DATA_BLOCK "InstEmDataHmi"   // DB44
TITLE = Instanz von FB EnergyMeterDataToHmi / Instance of FB instance of FB EnergyMeterDataToHmi
AUTHOR : SICAR
FAMILY : Energy
VERSION : 1.0
// Energy meter HMI
// stored: InstanceOfName LSicar_EnMeterDataToHmi, InstanceOfType FB
"LSicar_EnMeterDataToHmi"
   // VAR_INPUT
   //    energyMeter01Visu { ExternalAccessible := 'False'; ExternalVisible := 'False'; ExternalWritable := 'False'} : "LSicar_typeEnMeterVisuStruct";
   //    energyMeter02Visu { ExternalAccessible := 'False'; ExternalVisible := 'False'; ExternalWritable := 'False'} : "LSicar_typeEnMeterVisuStruct";
   //    energyMeter03Visu { ExternalAccessible := 'False'; ExternalVisible := 'False'; ExternalWritable := 'False'} : "LSicar_typeEnMeterVisuStruct";
   //    energyMeter04Visu { ExternalAccessible := 'False'; ExternalVisible := 'False'; ExternalWritable := 'False'} : "LSicar_typeEnMeterVisuStruct";
   //    energyMeter05Visu { ExternalAccessible := 'False'; ExternalVisible := 'False'; ExternalWritable := 'False'} : "LSicar_typeEnMeterVisuStruct";
   //    energyMeter06Visu { ExternalAccessible := 'False'; ExternalVisible := 'False'; ExternalWritable := 'False'} : "LSicar_typeEnMeterVisuStruct";
   //    energyMeter07Visu { ExternalAccessible := 'False'; ExternalVisible := 'False'; ExternalWritable := 'False'} : "LSicar_typeEnMeterVisuStruct";
   //    energyMeter08Visu { ExternalAccessible := 'False'; ExternalVisible := 'False'; ExternalWritable := 'False'} : "LSicar_typeEnMeterVisuStruct";
   // END_VAR
   // VAR
   //    statEmIndex : Int := 1;
   //    statEmData : "LSicar_typeEnMeterVisuStruct";
   //    statResetMinMaxAll : Bool := FALSE;
   //    statResetMinMax : Array[0..8] of Bool;
   //    statResetEnCounterAll : Bool := FALSE;
   //    statResetEnCounter : Array[0..8] of Bool;
   // END_VAR
BEGIN
   energyMeter01Visu.uL1L2 := 480.6464;
   energyMeter01Visu.uL2L3 := 479.3329;
   energyMeter01Visu.uL3L1 := 482.4024;
   energyMeter01Visu.uL1 := 277.0244;
   energyMeter01Visu.uL2 := 283.0648;
   energyMeter01Visu.uL3 := 272.9026;
   energyMeter01Visu.uL1L2Min := 470.1363;
   energyMeter01Visu.uL2L3Min := 469.0945;
   energyMeter01Visu.uL3L1Min := 472.4617;
   energyMeter01Visu.uL1Min := 271.5103;
   energyMeter01Visu.uL2Min := 277.1332;
   energyMeter01Visu.uL3Min := 267.6445;
   energyMeter01Visu.uL1L2Max := 486.0269;
   energyMeter01Visu.uL2L3Max := 484.8441;
   energyMeter01Visu.uL3L1Max := 487.8807;
   energyMeter01Visu.uL1Max := 280.1993;
   energyMeter01Visu.uL2Max := 286.2231;
   energyMeter01Visu.uL3Max := 276.0547;
   energyMeter01Visu.uPhPhAverage := 480.7939;
   energyMeter01Visu.uPhNaverage := 277.6639;
   energyMeter01Visu.uPhPhAverageMin := 470.5642;
   energyMeter01Visu.uPhNaverageMin := 272.105;
   energyMeter01Visu.uPhPhAverageMax := 486.2456;
   energyMeter01Visu.uPhNaverageMax := 280.8176;
   energyMeter01Visu.iL1 := 0.6297245;
   energyMeter01Visu.iL2 := 0.4116209;
   energyMeter01Visu.iL3 := 0.4021624;
   energyMeter01Visu.iL1Min := 0.5503862;
   energyMeter01Visu.iL2Min := 0.3512777;
   energyMeter01Visu.iL3Min := 0.3410119;
   energyMeter01Visu.iL1Max := 2.701323;
   energyMeter01Visu.iL2Max := 2.376321;
   energyMeter01Visu.iL3Max := 1.768756;
   energyMeter01Visu.iAverage := 0.4811693;
   energyMeter01Visu.iAverageMin := 0.4219982;
   energyMeter01Visu.iAverageMax := 2.194234;
   energyMeter01Visu.f := 59.99327;
   energyMeter01Visu.fMin := 59.9567;
   energyMeter01Visu.fMax := 60.07609;
   energyMeter01Visu.sTotal := 400.7156;
   energyMeter01Visu.sTotalMin := 349.7767;
   energyMeter01Visu.sTotalMax := 1823.43;
   energyMeter01Visu.pTotal := 277.3849;
   energyMeter01Visu.pTotalMin := 220.7085;
   energyMeter01Visu.pTotalMax := 670.0833;
   energyMeter01Visu.qTotal := -19.24654;
   energyMeter01Visu.qTotalMin := -422.0206;
   energyMeter01Visu.qTotalMax := -5.418034;
   energyMeter01Visu.cosL1 := 0.8610036;
   energyMeter01Visu.cosL1Min := 0.3576268;
   energyMeter01Visu.cosL1Max := 0.9157406;
   energyMeter01Visu.cosL2 := 0.5061908;
   energyMeter01Visu.cosL2Min := 0.05827232;
   energyMeter01Visu.cosL2Max := 0.7094496;
   energyMeter01Visu.cosL3 := 0.6214478;
   energyMeter01Visu.cosL3Min := 0.1665398;
   energyMeter01Visu.cosL3Max := 0.7301649;
   energyMeter01Visu.cosAverage := 0.6922238;
   energyMeter01Visu.cosAverageMin := 0.2474333;
   energyMeter01Visu.cosAverageMax := 0.7716895;
   energyMeter01Visu.sL1 := 174.449;
   energyMeter01Visu.sL2 := 116.5154;
   energyMeter01Visu.sL3 := 109.7511;
   energyMeter01Visu.sL1Min := 151.7066;
   energyMeter01Visu.sL2Min := 99.03358;
   energyMeter01Visu.sL3Min := 92.7289;
   energyMeter01Visu.sL1Max := 744.3881;
   energyMeter01Visu.sL2Max := 669.9091;
   energyMeter01Visu.sL3Max := 480.3434;
   energyMeter01Visu.pL1 := 150.2012;
   energyMeter01Visu.pL2 := 58.97903;
   energyMeter01Visu.pL3 := 68.20461;
   energyMeter01Visu.pL1Min := 127.6866;
   energyMeter01Visu.pL2Min := 20.87;
   energyMeter01Visu.pL3Min := 52.5906;
   energyMeter01Visu.pL1Max := 281.8818;
   energyMeter01Visu.pL2Max := 194.1828;
   energyMeter01Visu.pL3Max := 220.8245;
   energyMeter01Visu.qL1 := -4.041785;
   energyMeter01Visu.qL2 := 41.25737;
   energyMeter01Visu.qL3 := -56.46213;
   energyMeter01Visu.qL1Min := -144.4171;
   energyMeter01Visu.qL2Min := -98.00859;
   energyMeter01Visu.qL3Min := -198.8008;
   energyMeter01Visu.qL1Max := 28.71266;
   energyMeter01Visu.qL2Max := 50.3845;
   energyMeter01Visu.qL3Max := -53.43742;
   energyMeter01Visu.eActiveRate1Import := 736796.1;
   energyMeter01Visu.eActiveRate2Import := 0.0;
   energyMeter01Visu.eActiveRate1Export := 0.0002530577;
   energyMeter01Visu.eActiveRate2Export := 0.0;
   energyMeter01Visu.eReactiveRate1Import := 5676.457;
   energyMeter01Visu.eReactiveRate2Import := 0.0;
   energyMeter01Visu.eReactiveRate1Export := 293593.3;
   energyMeter01Visu.eReactiveRate2Export := 0.0;
   energyMeter01Visu.eApparentRate1Import := 1470773.0;
   energyMeter01Visu.eApparentRate2Import := 0.0;
   energyMeter01Visu.rTimeDataEnergy := DTL#1970-01-01-00:00:00;
   energyMeter01Visu.rTimeDataValue := DTL#1970-01-01-00:00:00;
   energyMeter01Visu.uPhPhMod := 16#0000;
   energyMeter01Visu.uPhNmod := 16#0000;
   energyMeter01Visu.iMod := 16#0000;
   energyMeter01Visu.sMod := 16#0000;
   energyMeter01Visu.pMod := 16#0000;
   energyMeter01Visu.qMod := 16#0000;
   energyMeter01Visu.eMod := 16#0000;
   energyMeter01Visu.fMod := 16#0000;
   energyMeter01Visu.cosMod := 16#0000;
   energyMeter01Visu.calculateValue1 := 16#0000;
   energyMeter01Visu.calculateValue2 := 16#0000;
   energyMeter01Visu.calculateValue3 := 16#0000;
   energyMeter01Visu.calculateValue4 := 16#0000;
   energyMeter01Visu.calculateValue5 := 16#0000;
   energyMeter01Visu.calculateValue6 := 16#0000;
   energyMeter01Visu.energyMeterUnit := 16#0000;
   energyMeter01Visu.restStartAuto := FALSE;
   energyMeter01Visu.readValue := FALSE;
   energyMeter01Visu.connectionType := 0;
   energyMeter01Visu.driverError := 0;
   energyMeter02Visu.uL1L2 := 0.0;
   energyMeter02Visu.uL2L3 := 0.0;
   energyMeter02Visu.uL3L1 := 0.0;
   energyMeter02Visu.uL1 := 0.0;
   energyMeter02Visu.uL2 := 0.0;
   energyMeter02Visu.uL3 := 0.0;
   energyMeter02Visu.uL1L2Min := 0.0;
   energyMeter02Visu.uL2L3Min := 0.0;
   energyMeter02Visu.uL3L1Min := 0.0;
   energyMeter02Visu.uL1Min := 0.0;
   energyMeter02Visu.uL2Min := 0.0;
   energyMeter02Visu.uL3Min := 0.0;
   energyMeter02Visu.uL1L2Max := 0.0;
   energyMeter02Visu.uL2L3Max := 0.0;
   energyMeter02Visu.uL3L1Max := 0.0;
   energyMeter02Visu.uL1Max := 0.0;
   energyMeter02Visu.uL2Max := 0.0;
   energyMeter02Visu.uL3Max := 0.0;
   energyMeter02Visu.uPhPhAverage := 0.0;
   energyMeter02Visu.uPhNaverage := 0.0;
   energyMeter02Visu.uPhPhAverageMin := 0.0;
   energyMeter02Visu.uPhNaverageMin := 0.0;
   energyMeter02Visu.uPhPhAverageMax := 0.0;
   energyMeter02Visu.uPhNaverageMax := 0.0;
   energyMeter02Visu.iL1 := 0.0;
   energyMeter02Visu.iL2 := 0.0;
   energyMeter02Visu.iL3 := 0.0;
   energyMeter02Visu.iL1Min := 0.0;
   energyMeter02Visu.iL2Min := 0.0;
   energyMeter02Visu.iL3Min := 0.0;
   energyMeter02Visu.iL1Max := 0.0;
   energyMeter02Visu.iL2Max := 0.0;
   energyMeter02Visu.iL3Max := 0.0;
   energyMeter02Visu.iAverage := 0.0;
   energyMeter02Visu.iAverageMin := 0.0;
   energyMeter02Visu.iAverageMax := 0.0;
   energyMeter02Visu.f := 0.0;
   energyMeter02Visu.fMin := 0.0;
   energyMeter02Visu.fMax := 0.0;
   energyMeter02Visu.sTotal := 0.0;
   energyMeter02Visu.sTotalMin := 0.0;
   energyMeter02Visu.sTotalMax := 0.0;
   energyMeter02Visu.pTotal := 0.0;
   energyMeter02Visu.pTotalMin := 0.0;
   energyMeter02Visu.pTotalMax := 0.0;
   energyMeter02Visu.qTotal := 0.0;
   energyMeter02Visu.qTotalMin := 0.0;
   energyMeter02Visu.qTotalMax := 0.0;
   energyMeter02Visu.cosL1 := 0.0;
   energyMeter02Visu.cosL1Min := 0.0;
   energyMeter02Visu.cosL1Max := 0.0;
   energyMeter02Visu.cosL2 := 0.0;
   energyMeter02Visu.cosL2Min := 0.0;
   energyMeter02Visu.cosL2Max := 0.0;
   energyMeter02Visu.cosL3 := 0.0;
   energyMeter02Visu.cosL3Min := 0.0;
   energyMeter02Visu.cosL3Max := 0.0;
   energyMeter02Visu.cosAverage := 0.0;
   energyMeter02Visu.cosAverageMin := 0.0;
   energyMeter02Visu.cosAverageMax := 0.0;
   energyMeter02Visu.sL1 := 0.0;
   energyMeter02Visu.sL2 := 0.0;
   energyMeter02Visu.sL3 := 0.0;
   energyMeter02Visu.sL1Min := 0.0;
   energyMeter02Visu.sL2Min := 0.0;
   energyMeter02Visu.sL3Min := 0.0;
   energyMeter02Visu.sL1Max := 0.0;
   energyMeter02Visu.sL2Max := 0.0;
   energyMeter02Visu.sL3Max := 0.0;
   energyMeter02Visu.pL1 := 0.0;
   energyMeter02Visu.pL2 := 0.0;
   energyMeter02Visu.pL3 := 0.0;
   energyMeter02Visu.pL1Min := 0.0;
   energyMeter02Visu.pL2Min := 0.0;
   energyMeter02Visu.pL3Min := 0.0;
   energyMeter02Visu.pL1Max := 0.0;
   energyMeter02Visu.pL2Max := 0.0;
   energyMeter02Visu.pL3Max := 0.0;
   energyMeter02Visu.qL1 := 0.0;
   energyMeter02Visu.qL2 := 0.0;
   energyMeter02Visu.qL3 := 0.0;
   energyMeter02Visu.qL1Min := 0.0;
   energyMeter02Visu.qL2Min := 0.0;
   energyMeter02Visu.qL3Min := 0.0;
   energyMeter02Visu.qL1Max := 0.0;
   energyMeter02Visu.qL2Max := 0.0;
   energyMeter02Visu.qL3Max := 0.0;
   energyMeter02Visu.eActiveRate1Import := 0.0;
   energyMeter02Visu.eActiveRate2Import := 0.0;
   energyMeter02Visu.eActiveRate1Export := 0.0;
   energyMeter02Visu.eActiveRate2Export := 0.0;
   energyMeter02Visu.eReactiveRate1Import := 0.0;
   energyMeter02Visu.eReactiveRate2Import := 0.0;
   energyMeter02Visu.eReactiveRate1Export := 0.0;
   energyMeter02Visu.eReactiveRate2Export := 0.0;
   energyMeter02Visu.eApparentRate1Import := 0.0;
   energyMeter02Visu.eApparentRate2Import := 0.0;
   energyMeter02Visu.rTimeDataEnergy := DTL#1970-01-01-00:00:00;
   energyMeter02Visu.rTimeDataValue := DTL#1970-01-01-00:00:00;
   energyMeter02Visu.uPhPhMod := 16#0000;
   energyMeter02Visu.uPhNmod := 16#0000;
   energyMeter02Visu.iMod := 16#0000;
   energyMeter02Visu.sMod := 16#0000;
   energyMeter02Visu.pMod := 16#0000;
   energyMeter02Visu.qMod := 16#0000;
   energyMeter02Visu.eMod := 16#0000;
   energyMeter02Visu.fMod := 16#0000;
   energyMeter02Visu.cosMod := 16#0000;
   energyMeter02Visu.calculateValue1 := 16#0000;
   energyMeter02Visu.calculateValue2 := 16#0000;
   energyMeter02Visu.calculateValue3 := 16#0000;
   energyMeter02Visu.calculateValue4 := 16#0000;
   energyMeter02Visu.calculateValue5 := 16#0000;
   energyMeter02Visu.calculateValue6 := 16#0000;
   energyMeter02Visu.energyMeterUnit := 16#0000;
   energyMeter02Visu.restStartAuto := FALSE;
   energyMeter02Visu.readValue := FALSE;
   energyMeter02Visu.connectionType := 0;
   energyMeter02Visu.driverError := 0;
   energyMeter03Visu.uL1L2 := 0.0;
   energyMeter03Visu.uL2L3 := 0.0;
   energyMeter03Visu.uL3L1 := 0.0;
   energyMeter03Visu.uL1 := 0.0;
   energyMeter03Visu.uL2 := 0.0;
   energyMeter03Visu.uL3 := 0.0;
   energyMeter03Visu.uL1L2Min := 0.0;
   energyMeter03Visu.uL2L3Min := 0.0;
   energyMeter03Visu.uL3L1Min := 0.0;
   energyMeter03Visu.uL1Min := 0.0;
   energyMeter03Visu.uL2Min := 0.0;
   energyMeter03Visu.uL3Min := 0.0;
   energyMeter03Visu.uL1L2Max := 0.0;
   energyMeter03Visu.uL2L3Max := 0.0;
   energyMeter03Visu.uL3L1Max := 0.0;
   energyMeter03Visu.uL1Max := 0.0;
   energyMeter03Visu.uL2Max := 0.0;
   energyMeter03Visu.uL3Max := 0.0;
   energyMeter03Visu.uPhPhAverage := 0.0;
   energyMeter03Visu.uPhNaverage := 0.0;
   energyMeter03Visu.uPhPhAverageMin := 0.0;
   energyMeter03Visu.uPhNaverageMin := 0.0;
   energyMeter03Visu.uPhPhAverageMax := 0.0;
   energyMeter03Visu.uPhNaverageMax := 0.0;
   energyMeter03Visu.iL1 := 0.0;
   energyMeter03Visu.iL2 := 0.0;
   energyMeter03Visu.iL3 := 0.0;
   energyMeter03Visu.iL1Min := 0.0;
   energyMeter03Visu.iL2Min := 0.0;
   energyMeter03Visu.iL3Min := 0.0;
   energyMeter03Visu.iL1Max := 0.0;
   energyMeter03Visu.iL2Max := 0.0;
   energyMeter03Visu.iL3Max := 0.0;
   energyMeter03Visu.iAverage := 0.0;
   energyMeter03Visu.iAverageMin := 0.0;
   energyMeter03Visu.iAverageMax := 0.0;
   energyMeter03Visu.f := 0.0;
   energyMeter03Visu.fMin := 0.0;
   energyMeter03Visu.fMax := 0.0;
   energyMeter03Visu.sTotal := 0.0;
   energyMeter03Visu.sTotalMin := 0.0;
   energyMeter03Visu.sTotalMax := 0.0;
   energyMeter03Visu.pTotal := 0.0;
   energyMeter03Visu.pTotalMin := 0.0;
   energyMeter03Visu.pTotalMax := 0.0;
   energyMeter03Visu.qTotal := 0.0;
   energyMeter03Visu.qTotalMin := 0.0;
   energyMeter03Visu.qTotalMax := 0.0;
   energyMeter03Visu.cosL1 := 0.0;
   energyMeter03Visu.cosL1Min := 0.0;
   energyMeter03Visu.cosL1Max := 0.0;
   energyMeter03Visu.cosL2 := 0.0;
   energyMeter03Visu.cosL2Min := 0.0;
   energyMeter03Visu.cosL2Max := 0.0;
   energyMeter03Visu.cosL3 := 0.0;
   energyMeter03Visu.cosL3Min := 0.0;
   energyMeter03Visu.cosL3Max := 0.0;
   energyMeter03Visu.cosAverage := 0.0;
   energyMeter03Visu.cosAverageMin := 0.0;
   energyMeter03Visu.cosAverageMax := 0.0;
   energyMeter03Visu.sL1 := 0.0;
   energyMeter03Visu.sL2 := 0.0;
   energyMeter03Visu.sL3 := 0.0;
   energyMeter03Visu.sL1Min := 0.0;
   energyMeter03Visu.sL2Min := 0.0;
   energyMeter03Visu.sL3Min := 0.0;
   energyMeter03Visu.sL1Max := 0.0;
   energyMeter03Visu.sL2Max := 0.0;
   energyMeter03Visu.sL3Max := 0.0;
   energyMeter03Visu.pL1 := 0.0;
   energyMeter03Visu.pL2 := 0.0;
   energyMeter03Visu.pL3 := 0.0;
   energyMeter03Visu.pL1Min := 0.0;
   energyMeter03Visu.pL2Min := 0.0;
   energyMeter03Visu.pL3Min := 0.0;
   energyMeter03Visu.pL1Max := 0.0;
   energyMeter03Visu.pL2Max := 0.0;
   energyMeter03Visu.pL3Max := 0.0;
   energyMeter03Visu.qL1 := 0.0;
   energyMeter03Visu.qL2 := 0.0;
   energyMeter03Visu.qL3 := 0.0;
   energyMeter03Visu.qL1Min := 0.0;
   energyMeter03Visu.qL2Min := 0.0;
   energyMeter03Visu.qL3Min := 0.0;
   energyMeter03Visu.qL1Max := 0.0;
   energyMeter03Visu.qL2Max := 0.0;
   energyMeter03Visu.qL3Max := 0.0;
   energyMeter03Visu.eActiveRate1Import := 0.0;
   energyMeter03Visu.eActiveRate2Import := 0.0;
   energyMeter03Visu.eActiveRate1Export := 0.0;
   energyMeter03Visu.eActiveRate2Export := 0.0;
   energyMeter03Visu.eReactiveRate1Import := 0.0;
   energyMeter03Visu.eReactiveRate2Import := 0.0;
   energyMeter03Visu.eReactiveRate1Export := 0.0;
   energyMeter03Visu.eReactiveRate2Export := 0.0;
   energyMeter03Visu.eApparentRate1Import := 0.0;
   energyMeter03Visu.eApparentRate2Import := 0.0;
   energyMeter03Visu.rTimeDataEnergy := DTL#1970-01-01-00:00:00;
   energyMeter03Visu.rTimeDataValue := DTL#1970-01-01-00:00:00;
   energyMeter03Visu.uPhPhMod := 16#0000;
   energyMeter03Visu.uPhNmod := 16#0000;
   energyMeter03Visu.iMod := 16#0000;
   energyMeter03Visu.sMod := 16#0000;
   energyMeter03Visu.pMod := 16#0000;
   energyMeter03Visu.qMod := 16#0000;
   energyMeter03Visu.eMod := 16#0000;
   energyMeter03Visu.fMod := 16#0000;
   energyMeter03Visu.cosMod := 16#0000;
   energyMeter03Visu.calculateValue1 := 16#0000;
   energyMeter03Visu.calculateValue2 := 16#0000;
   energyMeter03Visu.calculateValue3 := 16#0000;
   energyMeter03Visu.calculateValue4 := 16#0000;
   energyMeter03Visu.calculateValue5 := 16#0000;
   energyMeter03Visu.calculateValue6 := 16#0000;
   energyMeter03Visu.energyMeterUnit := 16#0000;
   energyMeter03Visu.restStartAuto := FALSE;
   energyMeter03Visu.readValue := FALSE;
   energyMeter03Visu.connectionType := 0;
   energyMeter03Visu.driverError := 0;
   energyMeter04Visu.uL1L2 := 0.0;
   energyMeter04Visu.uL2L3 := 0.0;
   energyMeter04Visu.uL3L1 := 0.0;
   energyMeter04Visu.uL1 := 0.0;
   energyMeter04Visu.uL2 := 0.0;
   energyMeter04Visu.uL3 := 0.0;
   energyMeter04Visu.uL1L2Min := 0.0;
   energyMeter04Visu.uL2L3Min := 0.0;
   energyMeter04Visu.uL3L1Min := 0.0;
   energyMeter04Visu.uL1Min := 0.0;
   energyMeter04Visu.uL2Min := 0.0;
   energyMeter04Visu.uL3Min := 0.0;
   energyMeter04Visu.uL1L2Max := 0.0;
   energyMeter04Visu.uL2L3Max := 0.0;
   energyMeter04Visu.uL3L1Max := 0.0;
   energyMeter04Visu.uL1Max := 0.0;
   energyMeter04Visu.uL2Max := 0.0;
   energyMeter04Visu.uL3Max := 0.0;
   energyMeter04Visu.uPhPhAverage := 0.0;
   energyMeter04Visu.uPhNaverage := 0.0;
   energyMeter04Visu.uPhPhAverageMin := 0.0;
   energyMeter04Visu.uPhNaverageMin := 0.0;
   energyMeter04Visu.uPhPhAverageMax := 0.0;
   energyMeter04Visu.uPhNaverageMax := 0.0;
   energyMeter04Visu.iL1 := 0.0;
   energyMeter04Visu.iL2 := 0.0;
   energyMeter04Visu.iL3 := 0.0;
   energyMeter04Visu.iL1Min := 0.0;
   energyMeter04Visu.iL2Min := 0.0;
   energyMeter04Visu.iL3Min := 0.0;
   energyMeter04Visu.iL1Max := 0.0;
   energyMeter04Visu.iL2Max := 0.0;
   energyMeter04Visu.iL3Max := 0.0;
   energyMeter04Visu.iAverage := 0.0;
   energyMeter04Visu.iAverageMin := 0.0;
   energyMeter04Visu.iAverageMax := 0.0;
   energyMeter04Visu.f := 0.0;
   energyMeter04Visu.fMin := 0.0;
   energyMeter04Visu.fMax := 0.0;
   energyMeter04Visu.sTotal := 0.0;
   energyMeter04Visu.sTotalMin := 0.0;
   energyMeter04Visu.sTotalMax := 0.0;
   energyMeter04Visu.pTotal := 0.0;
   energyMeter04Visu.pTotalMin := 0.0;
   energyMeter04Visu.pTotalMax := 0.0;
   energyMeter04Visu.qTotal := 0.0;
   energyMeter04Visu.qTotalMin := 0.0;
   energyMeter04Visu.qTotalMax := 0.0;
   energyMeter04Visu.cosL1 := 0.0;
   energyMeter04Visu.cosL1Min := 0.0;
   energyMeter04Visu.cosL1Max := 0.0;
   energyMeter04Visu.cosL2 := 0.0;
   energyMeter04Visu.cosL2Min := 0.0;
   energyMeter04Visu.cosL2Max := 0.0;
   energyMeter04Visu.cosL3 := 0.0;
   energyMeter04Visu.cosL3Min := 0.0;
   energyMeter04Visu.cosL3Max := 0.0;
   energyMeter04Visu.cosAverage := 0.0;
   energyMeter04Visu.cosAverageMin := 0.0;
   energyMeter04Visu.cosAverageMax := 0.0;
   energyMeter04Visu.sL1 := 0.0;
   energyMeter04Visu.sL2 := 0.0;
   energyMeter04Visu.sL3 := 0.0;
   energyMeter04Visu.sL1Min := 0.0;
   energyMeter04Visu.sL2Min := 0.0;
   energyMeter04Visu.sL3Min := 0.0;
   energyMeter04Visu.sL1Max := 0.0;
   energyMeter04Visu.sL2Max := 0.0;
   energyMeter04Visu.sL3Max := 0.0;
   energyMeter04Visu.pL1 := 0.0;
   energyMeter04Visu.pL2 := 0.0;
   energyMeter04Visu.pL3 := 0.0;
   energyMeter04Visu.pL1Min := 0.0;
   energyMeter04Visu.pL2Min := 0.0;
   energyMeter04Visu.pL3Min := 0.0;
   energyMeter04Visu.pL1Max := 0.0;
   energyMeter04Visu.pL2Max := 0.0;
   energyMeter04Visu.pL3Max := 0.0;
   energyMeter04Visu.qL1 := 0.0;
   energyMeter04Visu.qL2 := 0.0;
   energyMeter04Visu.qL3 := 0.0;
   energyMeter04Visu.qL1Min := 0.0;
   energyMeter04Visu.qL2Min := 0.0;
   energyMeter04Visu.qL3Min := 0.0;
   energyMeter04Visu.qL1Max := 0.0;
   energyMeter04Visu.qL2Max := 0.0;
   energyMeter04Visu.qL3Max := 0.0;
   energyMeter04Visu.eActiveRate1Import := 0.0;
   energyMeter04Visu.eActiveRate2Import := 0.0;
   energyMeter04Visu.eActiveRate1Export := 0.0;
   energyMeter04Visu.eActiveRate2Export := 0.0;
   energyMeter04Visu.eReactiveRate1Import := 0.0;
   energyMeter04Visu.eReactiveRate2Import := 0.0;
   energyMeter04Visu.eReactiveRate1Export := 0.0;
   energyMeter04Visu.eReactiveRate2Export := 0.0;
   energyMeter04Visu.eApparentRate1Import := 0.0;
   energyMeter04Visu.eApparentRate2Import := 0.0;
   energyMeter04Visu.rTimeDataEnergy := DTL#1970-01-01-00:00:00;
   energyMeter04Visu.rTimeDataValue := DTL#1970-01-01-00:00:00;
   energyMeter04Visu.uPhPhMod := 16#0000;
   energyMeter04Visu.uPhNmod := 16#0000;
   energyMeter04Visu.iMod := 16#0000;
   energyMeter04Visu.sMod := 16#0000;
   energyMeter04Visu.pMod := 16#0000;
   energyMeter04Visu.qMod := 16#0000;
   energyMeter04Visu.eMod := 16#0000;
   energyMeter04Visu.fMod := 16#0000;
   energyMeter04Visu.cosMod := 16#0000;
   energyMeter04Visu.calculateValue1 := 16#0000;
   energyMeter04Visu.calculateValue2 := 16#0000;
   energyMeter04Visu.calculateValue3 := 16#0000;
   energyMeter04Visu.calculateValue4 := 16#0000;
   energyMeter04Visu.calculateValue5 := 16#0000;
   energyMeter04Visu.calculateValue6 := 16#0000;
   energyMeter04Visu.energyMeterUnit := 16#0000;
   energyMeter04Visu.restStartAuto := FALSE;
   energyMeter04Visu.readValue := FALSE;
   energyMeter04Visu.connectionType := 0;
   energyMeter04Visu.driverError := 0;
   energyMeter05Visu.uL1L2 := 0.0;
   energyMeter05Visu.uL2L3 := 0.0;
   energyMeter05Visu.uL3L1 := 0.0;
   energyMeter05Visu.uL1 := 0.0;
   energyMeter05Visu.uL2 := 0.0;
   energyMeter05Visu.uL3 := 0.0;
   energyMeter05Visu.uL1L2Min := 0.0;
   energyMeter05Visu.uL2L3Min := 0.0;
   energyMeter05Visu.uL3L1Min := 0.0;
   energyMeter05Visu.uL1Min := 0.0;
   energyMeter05Visu.uL2Min := 0.0;
   energyMeter05Visu.uL3Min := 0.0;
   energyMeter05Visu.uL1L2Max := 0.0;
   energyMeter05Visu.uL2L3Max := 0.0;
   energyMeter05Visu.uL3L1Max := 0.0;
   energyMeter05Visu.uL1Max := 0.0;
   energyMeter05Visu.uL2Max := 0.0;
   energyMeter05Visu.uL3Max := 0.0;
   energyMeter05Visu.uPhPhAverage := 0.0;
   energyMeter05Visu.uPhNaverage := 0.0;
   energyMeter05Visu.uPhPhAverageMin := 0.0;
   energyMeter05Visu.uPhNaverageMin := 0.0;
   energyMeter05Visu.uPhPhAverageMax := 0.0;
   energyMeter05Visu.uPhNaverageMax := 0.0;
   energyMeter05Visu.iL1 := 0.0;
   energyMeter05Visu.iL2 := 0.0;
   energyMeter05Visu.iL3 := 0.0;
   energyMeter05Visu.iL1Min := 0.0;
   energyMeter05Visu.iL2Min := 0.0;
   energyMeter05Visu.iL3Min := 0.0;
   energyMeter05Visu.iL1Max := 0.0;
   energyMeter05Visu.iL2Max := 0.0;
   energyMeter05Visu.iL3Max := 0.0;
   energyMeter05Visu.iAverage := 0.0;
   energyMeter05Visu.iAverageMin := 0.0;
   energyMeter05Visu.iAverageMax := 0.0;
   energyMeter05Visu.f := 0.0;
   energyMeter05Visu.fMin := 0.0;
   energyMeter05Visu.fMax := 0.0;
   energyMeter05Visu.sTotal := 0.0;
   energyMeter05Visu.sTotalMin := 0.0;
   energyMeter05Visu.sTotalMax := 0.0;
   energyMeter05Visu.pTotal := 0.0;
   energyMeter05Visu.pTotalMin := 0.0;
   energyMeter05Visu.pTotalMax := 0.0;
   energyMeter05Visu.qTotal := 0.0;
   energyMeter05Visu.qTotalMin := 0.0;
   energyMeter05Visu.qTotalMax := 0.0;
   energyMeter05Visu.cosL1 := 0.0;
   energyMeter05Visu.cosL1Min := 0.0;
   energyMeter05Visu.cosL1Max := 0.0;
   energyMeter05Visu.cosL2 := 0.0;
   energyMeter05Visu.cosL2Min := 0.0;
   energyMeter05Visu.cosL2Max := 0.0;
   energyMeter05Visu.cosL3 := 0.0;
   energyMeter05Visu.cosL3Min := 0.0;
   energyMeter05Visu.cosL3Max := 0.0;
   energyMeter05Visu.cosAverage := 0.0;
   energyMeter05Visu.cosAverageMin := 0.0;
   energyMeter05Visu.cosAverageMax := 0.0;
   energyMeter05Visu.sL1 := 0.0;
   energyMeter05Visu.sL2 := 0.0;
   energyMeter05Visu.sL3 := 0.0;
   energyMeter05Visu.sL1Min := 0.0;
   energyMeter05Visu.sL2Min := 0.0;
   energyMeter05Visu.sL3Min := 0.0;
   energyMeter05Visu.sL1Max := 0.0;
   energyMeter05Visu.sL2Max := 0.0;
   energyMeter05Visu.sL3Max := 0.0;
   energyMeter05Visu.pL1 := 0.0;
   energyMeter05Visu.pL2 := 0.0;
   energyMeter05Visu.pL3 := 0.0;
   energyMeter05Visu.pL1Min := 0.0;
   energyMeter05Visu.pL2Min := 0.0;
   energyMeter05Visu.pL3Min := 0.0;
   energyMeter05Visu.pL1Max := 0.0;
   energyMeter05Visu.pL2Max := 0.0;
   energyMeter05Visu.pL3Max := 0.0;
   energyMeter05Visu.qL1 := 0.0;
   energyMeter05Visu.qL2 := 0.0;
   energyMeter05Visu.qL3 := 0.0;
   energyMeter05Visu.qL1Min := 0.0;
   energyMeter05Visu.qL2Min := 0.0;
   energyMeter05Visu.qL3Min := 0.0;
   energyMeter05Visu.qL1Max := 0.0;
   energyMeter05Visu.qL2Max := 0.0;
   energyMeter05Visu.qL3Max := 0.0;
   energyMeter05Visu.eActiveRate1Import := 0.0;
   energyMeter05Visu.eActiveRate2Import := 0.0;
   energyMeter05Visu.eActiveRate1Export := 0.0;
   energyMeter05Visu.eActiveRate2Export := 0.0;
   energyMeter05Visu.eReactiveRate1Import := 0.0;
   energyMeter05Visu.eReactiveRate2Import := 0.0;
   energyMeter05Visu.eReactiveRate1Export := 0.0;
   energyMeter05Visu.eReactiveRate2Export := 0.0;
   energyMeter05Visu.eApparentRate1Import := 0.0;
   energyMeter05Visu.eApparentRate2Import := 0.0;
   energyMeter05Visu.rTimeDataEnergy := DTL#1970-01-01-00:00:00;
   energyMeter05Visu.rTimeDataValue := DTL#1970-01-01-00:00:00;
   energyMeter05Visu.uPhPhMod := 16#0000;
   energyMeter05Visu.uPhNmod := 16#0000;
   energyMeter05Visu.iMod := 16#0000;
   energyMeter05Visu.sMod := 16#0000;
   energyMeter05Visu.pMod := 16#0000;
   energyMeter05Visu.qMod := 16#0000;
   energyMeter05Visu.eMod := 16#0000;
   energyMeter05Visu.fMod := 16#0000;
   energyMeter05Visu.cosMod := 16#0000;
   energyMeter05Visu.calculateValue1 := 16#0000;
   energyMeter05Visu.calculateValue2 := 16#0000;
   energyMeter05Visu.calculateValue3 := 16#0000;
   energyMeter05Visu.calculateValue4 := 16#0000;
   energyMeter05Visu.calculateValue5 := 16#0000;
   energyMeter05Visu.calculateValue6 := 16#0000;
   energyMeter05Visu.energyMeterUnit := 16#0000;
   energyMeter05Visu.restStartAuto := FALSE;
   energyMeter05Visu.readValue := FALSE;
   energyMeter05Visu.connectionType := 0;
   energyMeter05Visu.driverError := 0;
   energyMeter06Visu.uL1L2 := 0.0;
   energyMeter06Visu.uL2L3 := 0.0;
   energyMeter06Visu.uL3L1 := 0.0;
   energyMeter06Visu.uL1 := 0.0;
   energyMeter06Visu.uL2 := 0.0;
   energyMeter06Visu.uL3 := 0.0;
   energyMeter06Visu.uL1L2Min := 0.0;
   energyMeter06Visu.uL2L3Min := 0.0;
   energyMeter06Visu.uL3L1Min := 0.0;
   energyMeter06Visu.uL1Min := 0.0;
   energyMeter06Visu.uL2Min := 0.0;
   energyMeter06Visu.uL3Min := 0.0;
   energyMeter06Visu.uL1L2Max := 0.0;
   energyMeter06Visu.uL2L3Max := 0.0;
   energyMeter06Visu.uL3L1Max := 0.0;
   energyMeter06Visu.uL1Max := 0.0;
   energyMeter06Visu.uL2Max := 0.0;
   energyMeter06Visu.uL3Max := 0.0;
   energyMeter06Visu.uPhPhAverage := 0.0;
   energyMeter06Visu.uPhNaverage := 0.0;
   energyMeter06Visu.uPhPhAverageMin := 0.0;
   energyMeter06Visu.uPhNaverageMin := 0.0;
   energyMeter06Visu.uPhPhAverageMax := 0.0;
   energyMeter06Visu.uPhNaverageMax := 0.0;
   energyMeter06Visu.iL1 := 0.0;
   energyMeter06Visu.iL2 := 0.0;
   energyMeter06Visu.iL3 := 0.0;
   energyMeter06Visu.iL1Min := 0.0;
   energyMeter06Visu.iL2Min := 0.0;
   energyMeter06Visu.iL3Min := 0.0;
   energyMeter06Visu.iL1Max := 0.0;
   energyMeter06Visu.iL2Max := 0.0;
   energyMeter06Visu.iL3Max := 0.0;
   energyMeter06Visu.iAverage := 0.0;
   energyMeter06Visu.iAverageMin := 0.0;
   energyMeter06Visu.iAverageMax := 0.0;
   energyMeter06Visu.f := 0.0;
   energyMeter06Visu.fMin := 0.0;
   energyMeter06Visu.fMax := 0.0;
   energyMeter06Visu.sTotal := 0.0;
   energyMeter06Visu.sTotalMin := 0.0;
   energyMeter06Visu.sTotalMax := 0.0;
   energyMeter06Visu.pTotal := 0.0;
   energyMeter06Visu.pTotalMin := 0.0;
   energyMeter06Visu.pTotalMax := 0.0;
   energyMeter06Visu.qTotal := 0.0;
   energyMeter06Visu.qTotalMin := 0.0;
   energyMeter06Visu.qTotalMax := 0.0;
   energyMeter06Visu.cosL1 := 0.0;
   energyMeter06Visu.cosL1Min := 0.0;
   energyMeter06Visu.cosL1Max := 0.0;
   energyMeter06Visu.cosL2 := 0.0;
   energyMeter06Visu.cosL2Min := 0.0;
   energyMeter06Visu.cosL2Max := 0.0;
   energyMeter06Visu.cosL3 := 0.0;
   energyMeter06Visu.cosL3Min := 0.0;
   energyMeter06Visu.cosL3Max := 0.0;
   energyMeter06Visu.cosAverage := 0.0;
   energyMeter06Visu.cosAverageMin := 0.0;
   energyMeter06Visu.cosAverageMax := 0.0;
   energyMeter06Visu.sL1 := 0.0;
   energyMeter06Visu.sL2 := 0.0;
   energyMeter06Visu.sL3 := 0.0;
   energyMeter06Visu.sL1Min := 0.0;
   energyMeter06Visu.sL2Min := 0.0;
   energyMeter06Visu.sL3Min := 0.0;
   energyMeter06Visu.sL1Max := 0.0;
   energyMeter06Visu.sL2Max := 0.0;
   energyMeter06Visu.sL3Max := 0.0;
   energyMeter06Visu.pL1 := 0.0;
   energyMeter06Visu.pL2 := 0.0;
   energyMeter06Visu.pL3 := 0.0;
   energyMeter06Visu.pL1Min := 0.0;
   energyMeter06Visu.pL2Min := 0.0;
   energyMeter06Visu.pL3Min := 0.0;
   energyMeter06Visu.pL1Max := 0.0;
   energyMeter06Visu.pL2Max := 0.0;
   energyMeter06Visu.pL3Max := 0.0;
   energyMeter06Visu.qL1 := 0.0;
   energyMeter06Visu.qL2 := 0.0;
   energyMeter06Visu.qL3 := 0.0;
   energyMeter06Visu.qL1Min := 0.0;
   energyMeter06Visu.qL2Min := 0.0;
   energyMeter06Visu.qL3Min := 0.0;
   energyMeter06Visu.qL1Max := 0.0;
   energyMeter06Visu.qL2Max := 0.0;
   energyMeter06Visu.qL3Max := 0.0;
   energyMeter06Visu.eActiveRate1Import := 0.0;
   energyMeter06Visu.eActiveRate2Import := 0.0;
   energyMeter06Visu.eActiveRate1Export := 0.0;
   energyMeter06Visu.eActiveRate2Export := 0.0;
   energyMeter06Visu.eReactiveRate1Import := 0.0;
   energyMeter06Visu.eReactiveRate2Import := 0.0;
   energyMeter06Visu.eReactiveRate1Export := 0.0;
   energyMeter06Visu.eReactiveRate2Export := 0.0;
   energyMeter06Visu.eApparentRate1Import := 0.0;
   energyMeter06Visu.eApparentRate2Import := 0.0;
   energyMeter06Visu.rTimeDataEnergy := DTL#1970-01-01-00:00:00;
   energyMeter06Visu.rTimeDataValue := DTL#1970-01-01-00:00:00;
   energyMeter06Visu.uPhPhMod := 16#0000;
   energyMeter06Visu.uPhNmod := 16#0000;
   energyMeter06Visu.iMod := 16#0000;
   energyMeter06Visu.sMod := 16#0000;
   energyMeter06Visu.pMod := 16#0000;
   energyMeter06Visu.qMod := 16#0000;
   energyMeter06Visu.eMod := 16#0000;
   energyMeter06Visu.fMod := 16#0000;
   energyMeter06Visu.cosMod := 16#0000;
   energyMeter06Visu.calculateValue1 := 16#0000;
   energyMeter06Visu.calculateValue2 := 16#0000;
   energyMeter06Visu.calculateValue3 := 16#0000;
   energyMeter06Visu.calculateValue4 := 16#0000;
   energyMeter06Visu.calculateValue5 := 16#0000;
   energyMeter06Visu.calculateValue6 := 16#0000;
   energyMeter06Visu.energyMeterUnit := 16#0000;
   energyMeter06Visu.restStartAuto := FALSE;
   energyMeter06Visu.readValue := FALSE;
   energyMeter06Visu.connectionType := 0;
   energyMeter06Visu.driverError := 0;
   energyMeter07Visu.uL1L2 := 0.0;
   energyMeter07Visu.uL2L3 := 0.0;
   energyMeter07Visu.uL3L1 := 0.0;
   energyMeter07Visu.uL1 := 0.0;
   energyMeter07Visu.uL2 := 0.0;
   energyMeter07Visu.uL3 := 0.0;
   energyMeter07Visu.uL1L2Min := 0.0;
   energyMeter07Visu.uL2L3Min := 0.0;
   energyMeter07Visu.uL3L1Min := 0.0;
   energyMeter07Visu.uL1Min := 0.0;
   energyMeter07Visu.uL2Min := 0.0;
   energyMeter07Visu.uL3Min := 0.0;
   energyMeter07Visu.uL1L2Max := 0.0;
   energyMeter07Visu.uL2L3Max := 0.0;
   energyMeter07Visu.uL3L1Max := 0.0;
   energyMeter07Visu.uL1Max := 0.0;
   energyMeter07Visu.uL2Max := 0.0;
   energyMeter07Visu.uL3Max := 0.0;
   energyMeter07Visu.uPhPhAverage := 0.0;
   energyMeter07Visu.uPhNaverage := 0.0;
   energyMeter07Visu.uPhPhAverageMin := 0.0;
   energyMeter07Visu.uPhNaverageMin := 0.0;
   energyMeter07Visu.uPhPhAverageMax := 0.0;
   energyMeter07Visu.uPhNaverageMax := 0.0;
   energyMeter07Visu.iL1 := 0.0;
   energyMeter07Visu.iL2 := 0.0;
   energyMeter07Visu.iL3 := 0.0;
   energyMeter07Visu.iL1Min := 0.0;
   energyMeter07Visu.iL2Min := 0.0;
   energyMeter07Visu.iL3Min := 0.0;
   energyMeter07Visu.iL1Max := 0.0;
   energyMeter07Visu.iL2Max := 0.0;
   energyMeter07Visu.iL3Max := 0.0;
   energyMeter07Visu.iAverage := 0.0;
   energyMeter07Visu.iAverageMin := 0.0;
   energyMeter07Visu.iAverageMax := 0.0;
   energyMeter07Visu.f := 0.0;
   energyMeter07Visu.fMin := 0.0;
   energyMeter07Visu.fMax := 0.0;
   energyMeter07Visu.sTotal := 0.0;
   energyMeter07Visu.sTotalMin := 0.0;
   energyMeter07Visu.sTotalMax := 0.0;
   energyMeter07Visu.pTotal := 0.0;
   energyMeter07Visu.pTotalMin := 0.0;
   energyMeter07Visu.pTotalMax := 0.0;
   energyMeter07Visu.qTotal := 0.0;
   energyMeter07Visu.qTotalMin := 0.0;
   energyMeter07Visu.qTotalMax := 0.0;
   energyMeter07Visu.cosL1 := 0.0;
   energyMeter07Visu.cosL1Min := 0.0;
   energyMeter07Visu.cosL1Max := 0.0;
   energyMeter07Visu.cosL2 := 0.0;
   energyMeter07Visu.cosL2Min := 0.0;
   energyMeter07Visu.cosL2Max := 0.0;
   energyMeter07Visu.cosL3 := 0.0;
   energyMeter07Visu.cosL3Min := 0.0;
   energyMeter07Visu.cosL3Max := 0.0;
   energyMeter07Visu.cosAverage := 0.0;
   energyMeter07Visu.cosAverageMin := 0.0;
   energyMeter07Visu.cosAverageMax := 0.0;
   energyMeter07Visu.sL1 := 0.0;
   energyMeter07Visu.sL2 := 0.0;
   energyMeter07Visu.sL3 := 0.0;
   energyMeter07Visu.sL1Min := 0.0;
   energyMeter07Visu.sL2Min := 0.0;
   energyMeter07Visu.sL3Min := 0.0;
   energyMeter07Visu.sL1Max := 0.0;
   energyMeter07Visu.sL2Max := 0.0;
   energyMeter07Visu.sL3Max := 0.0;
   energyMeter07Visu.pL1 := 0.0;
   energyMeter07Visu.pL2 := 0.0;
   energyMeter07Visu.pL3 := 0.0;
   energyMeter07Visu.pL1Min := 0.0;
   energyMeter07Visu.pL2Min := 0.0;
   energyMeter07Visu.pL3Min := 0.0;
   energyMeter07Visu.pL1Max := 0.0;
   energyMeter07Visu.pL2Max := 0.0;
   energyMeter07Visu.pL3Max := 0.0;
   energyMeter07Visu.qL1 := 0.0;
   energyMeter07Visu.qL2 := 0.0;
   energyMeter07Visu.qL3 := 0.0;
   energyMeter07Visu.qL1Min := 0.0;
   energyMeter07Visu.qL2Min := 0.0;
   energyMeter07Visu.qL3Min := 0.0;
   energyMeter07Visu.qL1Max := 0.0;
   energyMeter07Visu.qL2Max := 0.0;
   energyMeter07Visu.qL3Max := 0.0;
   energyMeter07Visu.eActiveRate1Import := 0.0;
   energyMeter07Visu.eActiveRate2Import := 0.0;
   energyMeter07Visu.eActiveRate1Export := 0.0;
   energyMeter07Visu.eActiveRate2Export := 0.0;
   energyMeter07Visu.eReactiveRate1Import := 0.0;
   energyMeter07Visu.eReactiveRate2Import := 0.0;
   energyMeter07Visu.eReactiveRate1Export := 0.0;
   energyMeter07Visu.eReactiveRate2Export := 0.0;
   energyMeter07Visu.eApparentRate1Import := 0.0;
   energyMeter07Visu.eApparentRate2Import := 0.0;
   energyMeter07Visu.rTimeDataEnergy := DTL#1970-01-01-00:00:00;
   energyMeter07Visu.rTimeDataValue := DTL#1970-01-01-00:00:00;
   energyMeter07Visu.uPhPhMod := 16#0000;
   energyMeter07Visu.uPhNmod := 16#0000;
   energyMeter07Visu.iMod := 16#0000;
   energyMeter07Visu.sMod := 16#0000;
   energyMeter07Visu.pMod := 16#0000;
   energyMeter07Visu.qMod := 16#0000;
   energyMeter07Visu.eMod := 16#0000;
   energyMeter07Visu.fMod := 16#0000;
   energyMeter07Visu.cosMod := 16#0000;
   energyMeter07Visu.calculateValue1 := 16#0000;
   energyMeter07Visu.calculateValue2 := 16#0000;
   energyMeter07Visu.calculateValue3 := 16#0000;
   energyMeter07Visu.calculateValue4 := 16#0000;
   energyMeter07Visu.calculateValue5 := 16#0000;
   energyMeter07Visu.calculateValue6 := 16#0000;
   energyMeter07Visu.energyMeterUnit := 16#0000;
   energyMeter07Visu.restStartAuto := FALSE;
   energyMeter07Visu.readValue := FALSE;
   energyMeter07Visu.connectionType := 0;
   energyMeter07Visu.driverError := 0;
   energyMeter08Visu.uL1L2 := 0.0;
   energyMeter08Visu.uL2L3 := 0.0;
   energyMeter08Visu.uL3L1 := 0.0;
   energyMeter08Visu.uL1 := 0.0;
   energyMeter08Visu.uL2 := 0.0;
   energyMeter08Visu.uL3 := 0.0;
   energyMeter08Visu.uL1L2Min := 0.0;
   energyMeter08Visu.uL2L3Min := 0.0;
   energyMeter08Visu.uL3L1Min := 0.0;
   energyMeter08Visu.uL1Min := 0.0;
   energyMeter08Visu.uL2Min := 0.0;
   energyMeter08Visu.uL3Min := 0.0;
   energyMeter08Visu.uL1L2Max := 0.0;
   energyMeter08Visu.uL2L3Max := 0.0;
   energyMeter08Visu.uL3L1Max := 0.0;
   energyMeter08Visu.uL1Max := 0.0;
   energyMeter08Visu.uL2Max := 0.0;
   energyMeter08Visu.uL3Max := 0.0;
   energyMeter08Visu.uPhPhAverage := 0.0;
   energyMeter08Visu.uPhNaverage := 0.0;
   energyMeter08Visu.uPhPhAverageMin := 0.0;
   energyMeter08Visu.uPhNaverageMin := 0.0;
   energyMeter08Visu.uPhPhAverageMax := 0.0;
   energyMeter08Visu.uPhNaverageMax := 0.0;
   energyMeter08Visu.iL1 := 0.0;
   energyMeter08Visu.iL2 := 0.0;
   energyMeter08Visu.iL3 := 0.0;
   energyMeter08Visu.iL1Min := 0.0;
   energyMeter08Visu.iL2Min := 0.0;
   energyMeter08Visu.iL3Min := 0.0;
   energyMeter08Visu.iL1Max := 0.0;
   energyMeter08Visu.iL2Max := 0.0;
   energyMeter08Visu.iL3Max := 0.0;
   energyMeter08Visu.iAverage := 0.0;
   energyMeter08Visu.iAverageMin := 0.0;
   energyMeter08Visu.iAverageMax := 0.0;
   energyMeter08Visu.f := 0.0;
   energyMeter08Visu.fMin := 0.0;
   energyMeter08Visu.fMax := 0.0;
   energyMeter08Visu.sTotal := 0.0;
   energyMeter08Visu.sTotalMin := 0.0;
   energyMeter08Visu.sTotalMax := 0.0;
   energyMeter08Visu.pTotal := 0.0;
   energyMeter08Visu.pTotalMin := 0.0;
   energyMeter08Visu.pTotalMax := 0.0;
   energyMeter08Visu.qTotal := 0.0;
   energyMeter08Visu.qTotalMin := 0.0;
   energyMeter08Visu.qTotalMax := 0.0;
   energyMeter08Visu.cosL1 := 0.0;
   energyMeter08Visu.cosL1Min := 0.0;
   energyMeter08Visu.cosL1Max := 0.0;
   energyMeter08Visu.cosL2 := 0.0;
   energyMeter08Visu.cosL2Min := 0.0;
   energyMeter08Visu.cosL2Max := 0.0;
   energyMeter08Visu.cosL3 := 0.0;
   energyMeter08Visu.cosL3Min := 0.0;
   energyMeter08Visu.cosL3Max := 0.0;
   energyMeter08Visu.cosAverage := 0.0;
   energyMeter08Visu.cosAverageMin := 0.0;
   energyMeter08Visu.cosAverageMax := 0.0;
   energyMeter08Visu.sL1 := 0.0;
   energyMeter08Visu.sL2 := 0.0;
   energyMeter08Visu.sL3 := 0.0;
   energyMeter08Visu.sL1Min := 0.0;
   energyMeter08Visu.sL2Min := 0.0;
   energyMeter08Visu.sL3Min := 0.0;
   energyMeter08Visu.sL1Max := 0.0;
   energyMeter08Visu.sL2Max := 0.0;
   energyMeter08Visu.sL3Max := 0.0;
   energyMeter08Visu.pL1 := 0.0;
   energyMeter08Visu.pL2 := 0.0;
   energyMeter08Visu.pL3 := 0.0;
   energyMeter08Visu.pL1Min := 0.0;
   energyMeter08Visu.pL2Min := 0.0;
   energyMeter08Visu.pL3Min := 0.0;
   energyMeter08Visu.pL1Max := 0.0;
   energyMeter08Visu.pL2Max := 0.0;
   energyMeter08Visu.pL3Max := 0.0;
   energyMeter08Visu.qL1 := 0.0;
   energyMeter08Visu.qL2 := 0.0;
   energyMeter08Visu.qL3 := 0.0;
   energyMeter08Visu.qL1Min := 0.0;
   energyMeter08Visu.qL2Min := 0.0;
   energyMeter08Visu.qL3Min := 0.0;
   energyMeter08Visu.qL1Max := 0.0;
   energyMeter08Visu.qL2Max := 0.0;
   energyMeter08Visu.qL3Max := 0.0;
   energyMeter08Visu.eActiveRate1Import := 0.0;
   energyMeter08Visu.eActiveRate2Import := 0.0;
   energyMeter08Visu.eActiveRate1Export := 0.0;
   energyMeter08Visu.eActiveRate2Export := 0.0;
   energyMeter08Visu.eReactiveRate1Import := 0.0;
   energyMeter08Visu.eReactiveRate2Import := 0.0;
   energyMeter08Visu.eReactiveRate1Export := 0.0;
   energyMeter08Visu.eReactiveRate2Export := 0.0;
   energyMeter08Visu.eApparentRate1Import := 0.0;
   energyMeter08Visu.eApparentRate2Import := 0.0;
   energyMeter08Visu.rTimeDataEnergy := DTL#1970-01-01-00:00:00;
   energyMeter08Visu.rTimeDataValue := DTL#1970-01-01-00:00:00;
   energyMeter08Visu.uPhPhMod := 16#0000;
   energyMeter08Visu.uPhNmod := 16#0000;
   energyMeter08Visu.iMod := 16#0000;
   energyMeter08Visu.sMod := 16#0000;
   energyMeter08Visu.pMod := 16#0000;
   energyMeter08Visu.qMod := 16#0000;
   energyMeter08Visu.eMod := 16#0000;
   energyMeter08Visu.fMod := 16#0000;
   energyMeter08Visu.cosMod := 16#0000;
   energyMeter08Visu.calculateValue1 := 16#0000;
   energyMeter08Visu.calculateValue2 := 16#0000;
   energyMeter08Visu.calculateValue3 := 16#0000;
   energyMeter08Visu.calculateValue4 := 16#0000;
   energyMeter08Visu.calculateValue5 := 16#0000;
   energyMeter08Visu.calculateValue6 := 16#0000;
   energyMeter08Visu.energyMeterUnit := 16#0000;
   energyMeter08Visu.restStartAuto := FALSE;
   energyMeter08Visu.readValue := FALSE;
   energyMeter08Visu.connectionType := 0;
   energyMeter08Visu.driverError := 0;
   statEmData.uL1L2 := 480.6464;
   statEmData.uL2L3 := 479.3329;
   statEmData.uL3L1 := 482.4024;
   statEmData.uL1 := 277.0244;
   statEmData.uL2 := 283.0648;
   statEmData.uL3 := 272.9026;
   statEmData.uL1L2Min := 470.1363;
   statEmData.uL2L3Min := 469.0945;
   statEmData.uL3L1Min := 472.4617;
   statEmData.uL1Min := 271.5103;
   statEmData.uL2Min := 277.1332;
   statEmData.uL3Min := 267.6445;
   statEmData.uL1L2Max := 486.0269;
   statEmData.uL2L3Max := 484.8441;
   statEmData.uL3L1Max := 487.8807;
   statEmData.uL1Max := 280.1993;
   statEmData.uL2Max := 286.2231;
   statEmData.uL3Max := 276.0547;
   statEmData.uPhPhAverage := 480.7939;
   statEmData.uPhNaverage := 277.6639;
   statEmData.uPhPhAverageMin := 470.5642;
   statEmData.uPhNaverageMin := 272.105;
   statEmData.uPhPhAverageMax := 486.2456;
   statEmData.uPhNaverageMax := 280.8176;
   statEmData.iL1 := 0.6297245;
   statEmData.iL2 := 0.4116209;
   statEmData.iL3 := 0.4021624;
   statEmData.iL1Min := 0.5503862;
   statEmData.iL2Min := 0.3512777;
   statEmData.iL3Min := 0.3410119;
   statEmData.iL1Max := 2.701323;
   statEmData.iL2Max := 2.376321;
   statEmData.iL3Max := 1.768756;
   statEmData.iAverage := 0.4811693;
   statEmData.iAverageMin := 0.4219982;
   statEmData.iAverageMax := 2.194234;
   statEmData.f := 59.99327;
   statEmData.fMin := 59.9567;
   statEmData.fMax := 60.07609;
   statEmData.sTotal := 400.7156;
   statEmData.sTotalMin := 349.7767;
   statEmData.sTotalMax := 1823.43;
   statEmData.pTotal := 277.3849;
   statEmData.pTotalMin := 220.7085;
   statEmData.pTotalMax := 670.0833;
   statEmData.qTotal := -19.24654;
   statEmData.qTotalMin := -422.0206;
   statEmData.qTotalMax := -5.418034;
   statEmData.cosL1 := 0.8610036;
   statEmData.cosL1Min := 0.3576268;
   statEmData.cosL1Max := 0.9157406;
   statEmData.cosL2 := 0.5061908;
   statEmData.cosL2Min := 0.05827232;
   statEmData.cosL2Max := 0.7094496;
   statEmData.cosL3 := 0.6214478;
   statEmData.cosL3Min := 0.1665398;
   statEmData.cosL3Max := 0.7301649;
   statEmData.cosAverage := 0.6922238;
   statEmData.cosAverageMin := 0.2474333;
   statEmData.cosAverageMax := 0.7716895;
   statEmData.sL1 := 174.449;
   statEmData.sL2 := 116.5154;
   statEmData.sL3 := 109.7511;
   statEmData.sL1Min := 151.7066;
   statEmData.sL2Min := 99.03358;
   statEmData.sL3Min := 92.7289;
   statEmData.sL1Max := 744.3881;
   statEmData.sL2Max := 669.9091;
   statEmData.sL3Max := 480.3434;
   statEmData.pL1 := 150.2012;
   statEmData.pL2 := 58.97903;
   statEmData.pL3 := 68.20461;
   statEmData.pL1Min := 127.6866;
   statEmData.pL2Min := 20.87;
   statEmData.pL3Min := 52.5906;
   statEmData.pL1Max := 281.8818;
   statEmData.pL2Max := 194.1828;
   statEmData.pL3Max := 220.8245;
   statEmData.qL1 := -4.041785;
   statEmData.qL2 := 41.25737;
   statEmData.qL3 := -56.46213;
   statEmData.qL1Min := -144.4171;
   statEmData.qL2Min := -98.00859;
   statEmData.qL3Min := -198.8008;
   statEmData.qL1Max := 28.71266;
   statEmData.qL2Max := 50.3845;
   statEmData.qL3Max := -53.43742;
   statEmData.eActiveRate1Import := 736796.1;
   statEmData.eActiveRate2Import := 0.0;
   statEmData.eActiveRate1Export := 0.0002530577;
   statEmData.eActiveRate2Export := 0.0;
   statEmData.eReactiveRate1Import := 5676.457;
   statEmData.eReactiveRate2Import := 0.0;
   statEmData.eReactiveRate1Export := 293593.3;
   statEmData.eReactiveRate2Export := 0.0;
   statEmData.eApparentRate1Import := 1470773.0;
   statEmData.eApparentRate2Import := 0.0;
   statEmData.rTimeDataEnergy := DTL#1970-01-01-00:00:00;
   statEmData.rTimeDataValue := DTL#1970-01-01-00:00:00;
   statEmData.uPhPhMod := 16#0000;
   statEmData.uPhNmod := 16#0000;
   statEmData.iMod := 16#0000;
   statEmData.sMod := 16#0000;
   statEmData.pMod := 16#0000;
   statEmData.qMod := 16#0000;
   statEmData.eMod := 16#0000;
   statEmData.fMod := 16#0000;
   statEmData.cosMod := 16#0000;
   statEmData.calculateValue1 := 16#0000;
   statEmData.calculateValue2 := 16#0000;
   statEmData.calculateValue3 := 16#0000;
   statEmData.calculateValue4 := 16#0000;
   statEmData.calculateValue5 := 16#0000;
   statEmData.calculateValue6 := 16#0000;
   statEmData.energyMeterUnit := 16#0000;
   statEmData.restStartAuto := FALSE;
   statEmData.readValue := FALSE;
   statEmData.connectionType := 0;
   statEmData.driverError := 0;
   statResetMinMax[0..8] := FALSE;
   statResetEnCounter[0..8] := FALSE;
END_DATA_BLOCK

DATA_BLOCK "InstPlantSimulationTimer"   // DB110
{ DB_Accessible_From_OPC_UA := 'FALSE' }
// stored: DBAccessibleFromOPCUA false, DBAccessibleFromWebserver false, InstanceOfName IEC_TIMER, OfSystemLibElement IEC_TIMER, OfSystemLibVersion 1.0
"IEC_TIMER"
   // VAR
   //    PT : Time := T#0MS;
   //    ET { ExternalWritable := 'False'} : Time;
   //    IN : Bool := FALSE;
   //    Q { ExternalWritable := 'False'} : Bool;
   // END_VAR
BEGIN
END_DATA_BLOCK

DATA_BLOCK "InstSimulationTimer"   // DB111
TITLE = Simulation timer
// Instanz of IEC timer / instance of IEC timer
// stored: InstanceOfName IEC_TIMER, OfSystemLibElement IEC_TIMER, OfSystemLibVersion 1.0
"IEC_TIMER"
   // VAR
   //    PT : Time := T#0MS;
   //    ET { ExternalWritable := 'False'} : Time;
   //    IN : Bool := FALSE;
   //    Q { ExternalWritable := 'False'} : Bool;
   // END_VAR
BEGIN
END_DATA_BLOCK

DATA_BLOCK "InstSleepModeManager"   // DB488
// stored: InstanceOfName LER_SleepModeManager, InstanceOfType FB
"LER_SleepModeManager"
   // VAR_INPUT
   //    enable : Bool;
   //    unitStatus : "LAF_typeUnitStatus";
   //    wakeUpReq : Bool;
   //    sleepDelay : Time;
   //    deepSleepDelay : Time;
   // END_VAR
   // VAR_OUTPUT
   //    sleepModeChangeReq : Bool;
   //    deepSleepModeChangeReq : Bool;
   //    wakeUpRecoveryRequired : Bool;
   // END_VAR
   // VAR
   //    instSleepDelay { ExternalAccessible := 'False'; ExternalVisible := 'False'; ExternalWritable := 'False'; S7_SetPoint := 'True'} : TON_TIME;
   //    instDeepSleepDelay { ExternalAccessible := 'False'; ExternalVisible := 'False'; ExternalWritable := 'False'; S7_SetPoint := 'True'} : TON_TIME;
   //    statStandbyReady { ExternalAccessible := 'False'; ExternalVisible := 'False'; ExternalWritable := 'False'} : Bool;
   //    statWakeUpRecoveryRequired { ExternalAccessible := 'False'; ExternalVisible := 'False'; ExternalWritable := 'False'} : Bool;
   // END_VAR
BEGIN
END_DATA_BLOCK

DATA_BLOCK "InstChecksum"   // DB50
AUTHOR : SICAR
FAMILY : Diag
// stored: AssignedProDiagFB ProDiag, InstanceOfName LAF_Checksum, InstanceOfType FB
"LAF_Checksum"
   // VAR_INPUT
   //    plantIdentifier { ExternalAccessible := 'False'; ExternalVisible := 'False'; ExternalWritable := 'False'} : WString[24] := WSTRING#'PLC-Checksum';
   //    textListId { ExternalAccessible := 'False'; ExternalVisible := 'False'; ExternalWritable := 'False'} : Int := 584;
   //    dateTime { ExternalAccessible := 'False'; ExternalVisible := 'False'; ExternalWritable := 'False'} : Date_And_Time := DT#2026-01-06-19:57:41.039;
   //    readChecksum { ExternalAccessible := 'False'; ExternalVisible := 'False'; ExternalWritable := 'False'} : Bool := TRUE;
   //    ack { ExternalAccessible := 'False'; ExternalVisible := 'False'; ExternalWritable := 'False'} : Bool := FALSE;
   //    hideMessageStandard { ExternalAccessible := 'False'; ExternalVisible := 'False'; ExternalWritable := 'False'} : Bool := FALSE;
   //    hideMessageSafety { ExternalAccessible := 'False'; ExternalVisible := 'False'; ExternalWritable := 'False'} : Bool := FALSE;
   //    hideMessageTextlist { ExternalAccessible := 'False'; ExternalVisible := 'False'; ExternalWritable := 'False'} : Bool := FALSE;
   // END_VAR
   // VAR_OUTPUT
   //    generalMessage { ExternalAccessible := 'False'; ExternalVisible := 'False'; ExternalWritable := 'False'} : Bool := FALSE;
   // END_VAR
   // VAR_IN_OUT
   //    checksumHmi : "LAF_typeChecksum";
   // END_VAR
   // VAR
   //    statReadChecksumStorage { ExternalAccessible := 'False'; ExternalVisible := 'False'; ExternalWritable := 'False'} : Bool := FALSE;
   //    statChecksumStandard { ExternalAccessible := 'False'; ExternalVisible := 'False'; ExternalWritable := 'False'} : Array[0..7] of Byte;
   //    statChecksumStafety { ExternalAccessible := 'False'; ExternalVisible := 'False'; ExternalWritable := 'False'} : Array[0..7] of Byte;
   //    statChecksumTextlists { ExternalAccessible := 'False'; ExternalVisible := 'False'; ExternalWritable := 'False'} : Array[0..7] of Byte;
   //    statChecksumStandOldNull { ExternalAccessible := 'False'; ExternalVisible := 'False'; ExternalWritable := 'False'} : Bool := FALSE;
   //    statChecksumSafeOldNull { ExternalAccessible := 'False'; ExternalVisible := 'False'; ExternalWritable := 'False'} : Bool := FALSE;
   //    statChecksumTextlOldNull { ExternalAccessible := 'False'; ExternalVisible := 'False'; ExternalWritable := 'False'} : Bool := FALSE;
   //    statChecksumStandDiff { ExternalAccessible := 'False'; ExternalVisible := 'False'; ExternalWritable := 'False'} : Bool := FALSE;
   //    statChecksumSafeDiff { ExternalAccessible := 'False'; ExternalVisible := 'False'; ExternalWritable := 'False'} : Bool := FALSE;
   //    statChecksumTextlDiff { ExternalAccessible := 'False'; ExternalVisible := 'False'; ExternalWritable := 'False'} : Bool := FALSE;
   //    instGetChecksum1 { ExternalAccessible := 'False'; ExternalVisible := 'False'; ExternalWritable := 'False'} : GetChecksum;
   //    instGetChecksum2 { ExternalAccessible := 'False'; ExternalVisible := 'False'; ExternalWritable := 'False'} : GetChecksum;
   //    instGetChecksum3 { ExternalAccessible := 'False'; ExternalVisible := 'False'; ExternalWritable := 'False'} : GetChecksum;
   //    statRetValHta { ExternalAccessible := 'False'; ExternalVisible := 'False'; ExternalWritable := 'False'} : "LAF_typeChecksumCatWord";
   //    statRisEdgeDiff { ExternalAccessible := 'False'; ExternalVisible := 'False'; ExternalWritable := 'False'} : "LAF_typeChecksumCatBool";
   //    statMessageStandModified { ExternalAccessible := 'False'; ExternalVisible := 'False'; ExternalWritable := 'False'} : Bool := FALSE;
   //    statMessageSafeModified { ExternalAccessible := 'False'; ExternalVisible := 'False'; ExternalWritable := 'False'} : Bool := FALSE;
   //    statMessageTextlModified { ExternalAccessible := 'False'; ExternalVisible := 'False'; ExternalWritable := 'False'} : Bool := FALSE;
   //    statWarnNoStandard { ExternalAccessible := 'False'; ExternalVisible := 'False'; ExternalWritable := 'False'} : UInt := 99;
   //    statWarnNoSafety { ExternalAccessible := 'False'; ExternalVisible := 'False'; ExternalWritable := 'False'} : UInt := 99;
   //    statWarnNoTextlist { ExternalAccessible := 'False'; ExternalVisible := 'False'; ExternalWritable := 'False'} : UInt := 99;
   // END_VAR
BEGIN
   statChecksumStandard[0] := 16#E4;
   statChecksumStandard[1] := 16#AA;
   statChecksumStandard[2] := 16#23;
   statChecksumStandard[3] := 16#DF;
   statChecksumStandard[4] := 16#FD;
   statChecksumStandard[5] := 16#EE;
   statChecksumStandard[6] := 16#A8;
   statChecksumStandard[7] := 16#66;
   statChecksumStafety[0] := 16#0A;
   statChecksumStafety[1] := 16#6C;
   statChecksumStafety[2] := 16#EC;
   statChecksumStafety[3] := 16#4B;
   statChecksumStafety[4..7] := 16#00;
   statChecksumTextlists[0] := 16#67;
   statChecksumTextlists[1] := 16#6D;
   statChecksumTextlists[2] := 16#C4;
   statChecksumTextlists[3] := 16#50;
   statChecksumTextlists[4] := 16#55;
   statChecksumTextlists[5] := 16#90;
   statChecksumTextlists[6] := 16#21;
   statChecksumTextlists[7] := 16#79;
   instGetChecksum1.Scope := 1;
   instGetChecksum1.Done := TRUE;
   instGetChecksum1.Busy := FALSE;
   instGetChecksum1.Error := FALSE;
   instGetChecksum1.Status := 16#0000;
   instGetChecksum1.tmpNulled[0] := 16#E4;
   instGetChecksum1.tmpNulled[1] := 16#AA;
   instGetChecksum1.tmpNulled[2] := 16#23;
   instGetChecksum1.tmpNulled[3] := 16#DF;
   instGetChecksum1.tmpNulled[4] := 16#FD;
   instGetChecksum1.tmpNulled[5] := 16#EE;
   instGetChecksum1.tmpNulled[6] := 16#A8;
   instGetChecksum1.tmpNulled[7] := 16#66;
   instGetChecksum1.GMACount := 1;
   instGetChecksum1.GMAPathLens[0] := 3;
   instGetChecksum1.GMAPaths[0] := 16#89A0_0003;
   instGetChecksum1.GMAPaths[1] := 16#0000_1FC9;
   instGetChecksum1.GMAPaths[2] := 16#0000_0001;
   instGetChecksum1.GMAResLens[0] := 8;
   instGetChecksum2.Scope := 2;
   instGetChecksum2.Done := TRUE;
   instGetChecksum2.Busy := FALSE;
   instGetChecksum2.Error := FALSE;
   instGetChecksum2.Status := 16#0000;
   instGetChecksum2.tmpNulled[0] := 16#0A;
   instGetChecksum2.tmpNulled[1] := 16#6C;
   instGetChecksum2.tmpNulled[2] := 16#EC;
   instGetChecksum2.tmpNulled[3] := 16#4B;
   instGetChecksum2.tmpNulled[4..7] := 16#00;
   instGetChecksum2.GMACount := 1;
   instGetChecksum2.GMAPathLens[0] := 2;
   instGetChecksum2.GMAPaths[0] := 16#89F9_0000;
   instGetChecksum2.GMAPaths[1] := 16#0000_1E37;
   instGetChecksum2.GMAPaths[2] := 16#0000_0000;
   instGetChecksum2.GMAResLens[0] := 4;
   instGetChecksum3.Scope := 3;
   instGetChecksum3.Done := TRUE;
   instGetChecksum3.Busy := FALSE;
   instGetChecksum3.Error := FALSE;
   instGetChecksum3.Status := 16#0000;
   instGetChecksum3.tmpNulled[0] := 16#67;
   instGetChecksum3.tmpNulled[1] := 16#6D;
   instGetChecksum3.tmpNulled[2] := 16#C4;
   instGetChecksum3.tmpNulled[3] := 16#50;
   instGetChecksum3.tmpNulled[4] := 16#55;
   instGetChecksum3.tmpNulled[5] := 16#90;
   instGetChecksum3.tmpNulled[6] := 16#21;
   instGetChecksum3.tmpNulled[7] := 16#79;
   instGetChecksum3.GMACount := 1;
   instGetChecksum3.GMAPathLens[0] := 3;
   instGetChecksum3.GMAPaths[0] := 16#89A0_0072;
   instGetChecksum3.GMAPaths[1] := 16#0000_1FC9;
   instGetChecksum3.GMAPaths[2] := 16#0000_0001;
   instGetChecksum3.GMAResLens[0] := 8;
   statRetValHta.standard := 16#0000;
   statRetValHta.safety := 16#0000;
   statRetValHta.textlists := 16#0000;
   statRisEdgeDiff.standard := FALSE;
   statRisEdgeDiff.safety := FALSE;
   statRisEdgeDiff.textlists := FALSE;
END_DATA_BLOCK

DATA_BLOCK "InstMemCardDiag"   // DB122
AUTHOR : Siemens Digital Industries
FAMILY : LAF
// stored: AssignedProDiagFB ProDiag, InstanceOfName LAF_MemCardDiag, InstanceOfType FB
"LAF_MemCardDiag"
   // VAR_INPUT
   //    plantIdentifier { ExternalAccessible := 'False'; ExternalVisible := 'False'; ExternalWritable := 'False'} : WString[24] := WSTRING#'SMC_Diagnostic';
   //    textListId { ExternalAccessible := 'False'; ExternalVisible := 'False'; ExternalWritable := 'False'} : Int := 585;
   //    firstCycle { ExternalAccessible := 'False'; ExternalVisible := 'False'; ExternalWritable := 'False'} : Bool := FALSE;
   //    readInfoMemCard { ExternalAccessible := 'False'; ExternalVisible := 'False'; ExternalWritable := 'False'} : Bool := FALSE;
   //    hideAlarmMask { ExternalAccessible := 'False'; ExternalVisible := 'False'; ExternalWritable := 'False'} : Byte := 16#00;
   // END_VAR
   // VAR_OUTPUT
   //    generalAlarm { ExternalAccessible := 'False'; ExternalVisible := 'False'; ExternalWritable := 'False'} : Bool := FALSE;
   //    generalWarn { ExternalAccessible := 'False'; ExternalVisible := 'False'; ExternalWritable := 'False'} : Bool := FALSE;
   //    generalInfo { ExternalAccessible := 'False'; ExternalVisible := 'False'; ExternalWritable := 'False'} : Bool := FALSE;
   // END_VAR
   // VAR_IN_OUT
   //    diagHmi : "LAF_typeMemCardDiag";
   // END_VAR
   // VAR
   //    statMessages { ExternalAccessible := 'False'; ExternalVisible := 'False'; ExternalWritable := 'False'} : "LAF_typeMemCardMessages";
   //    statHideMessages { ExternalAccessible := 'False'; ExternalVisible := 'False'; ExternalWritable := 'False'} : "LAF_typeMemCardMessages";
   //    statStep { ExternalAccessible := 'False'; ExternalVisible := 'False'; ExternalWritable := 'False'} : Array[0..3] of Bool;
   //    statRisEdgeStep0 { ExternalAccessible := 'False'; ExternalVisible := 'False'; ExternalWritable := 'False'} : Bool := FALSE;
   //    statRisEdgeStep1 { ExternalAccessible := 'False'; ExternalVisible := 'False'; ExternalWritable := 'False'} : Bool := FALSE;
   //    statAlarmNo { ExternalAccessible := 'False'; ExternalVisible := 'False'; ExternalWritable := 'False'} : UInt := 99;
   //    statWarnNo { ExternalAccessible := 'False'; ExternalVisible := 'False'; ExternalWritable := 'False'} : UInt := 99;
   //    statInfoNo { ExternalAccessible := 'False'; ExternalVisible := 'False'; ExternalWritable := 'False'} : UInt := 99;
   //    instGetInfoMode0 { ExternalAccessible := 'False'; ExternalVisible := 'False'; ExternalWritable := 'False'} : GetSMCinfo;
   //    instGetInfoMode1 { ExternalAccessible := 'False'; ExternalVisible := 'False'; ExternalWritable := 'False'} : GetSMCinfo;
   //    instGetInfoMode2 { ExternalAccessible := 'False'; ExternalVisible := 'False'; ExternalWritable := 'False'} : GetSMCinfo;
   //    instGetInfoMode3 { ExternalAccessible := 'False'; ExternalVisible := 'False'; ExternalWritable := 'False'} : GetSMCinfo;
   // END_VAR
BEGIN
   statMessages.invalidValueModeParam := FALSE;
   statMessages.noMemCardInserted := FALSE;
   statMessages.noDataAvailable := FALSE;
   statMessages.maxCallsReached := FALSE;
   statMessages.configMemSpaceWarning := FALSE;
   statMessages.configMemSpaceAlarm := FALSE;
   statMessages.usedLiftetimeInvalid := FALSE;
   statMessages.diagAlarmDisabled := FALSE;
   statHideMessages.invalidValueModeParam := FALSE;
   statHideMessages.noMemCardInserted := FALSE;
   statHideMessages.noDataAvailable := FALSE;
   statHideMessages.maxCallsReached := FALSE;
   statHideMessages.configMemSpaceWarning := FALSE;
   statHideMessages.configMemSpaceAlarm := FALSE;
   statHideMessages.usedLiftetimeInvalid := FALSE;
   statHideMessages.diagAlarmDisabled := FALSE;
   statStep[0..3] := FALSE;
   instGetInfoMode0.REQ := FALSE;
   instGetInfoMode0.Mode := 0;
   instGetInfoMode0.Done := FALSE;
   instGetInfoMode0.Busy := FALSE;
   instGetInfoMode0.Error := FALSE;
   instGetInfoMode0.Status := 16#7000;
   instGetInfoMode0.Info := 31151664;
   instGetInfoMode1.REQ := FALSE;
   instGetInfoMode1.Mode := 1;
   instGetInfoMode1.Done := FALSE;
   instGetInfoMode1.Busy := FALSE;
   instGetInfoMode1.Error := FALSE;
   instGetInfoMode1.Status := 16#7000;
   instGetInfoMode1.Info := 68208;
   instGetInfoMode2.REQ := FALSE;
   instGetInfoMode2.Mode := 2;
   instGetInfoMode2.Done := FALSE;
   instGetInfoMode2.Busy := FALSE;
   instGetInfoMode2.Error := FALSE;
   instGetInfoMode2.Status := 16#7000;
   instGetInfoMode2.Info := 0;
   instGetInfoMode3.REQ := FALSE;
   instGetInfoMode3.Mode := 3;
   instGetInfoMode3.Done := FALSE;
   instGetInfoMode3.Busy := FALSE;
   instGetInfoMode3.Error := FALSE;
   instGetInfoMode3.Status := 16#7000;
   instGetInfoMode3.Info := 80;
END_DATA_BLOCK

DATA_BLOCK "InstPlcDiag"   // DB34
AUTHOR : Siemens Digital Industries
FAMILY : LAF
// stored: InstanceOfName LAF_PlcDiag, InstanceOfType FB
"LAF_PlcDiag"
   // VAR_INPUT
   //    localCommon { ExternalAccessible := 'False'; ExternalVisible := 'False'; ExternalWritable := 'False'} : HW_SUBMODULE := 50;
   //    localProfinetInterface { ExternalAccessible := 'False'; ExternalVisible := 'False'; ExternalWritable := 'False'} : HW_INTERFACE := 64;
   //    firstCycle { ExternalAccessible := 'False'; ExternalVisible := 'False'; ExternalWritable := 'False'} : Bool := FALSE;
   // END_VAR
   // VAR_IN_OUT
   //    diagDataHmi : "LAF_typePlcDiag";
   // END_VAR
   // VAR
   //    statLocalCommon { ExternalAccessible := 'False'; ExternalVisible := 'False'; ExternalWritable := 'False'} : HW_SUBMODULE := 50;
   //    statLocProfinetInterface { ExternalAccessible := 'False'; ExternalVisible := 'False'; ExternalWritable := 'False'} : HW_INTERFACE := 64;
   //    instGetImData0 { ExternalAccessible := 'False'; ExternalVisible := 'False'; ExternalWritable := 'False'} : Get_IM_Data;
   //    statGetImData0ErrorSaved { ExternalAccessible := 'False'; ExternalVisible := 'False'; ExternalWritable := 'False'} : Word := 16#0000;
   //    instGetImData1 { ExternalAccessible := 'False'; ExternalVisible := 'False'; ExternalWritable := 'False'} : Get_IM_Data;
   //    statGetImData1ErrorSaved { ExternalAccessible := 'False'; ExternalVisible := 'False'; ExternalWritable := 'False'} : Word := 16#0000;
   //    instGetImData2 { ExternalAccessible := 'False'; ExternalVisible := 'False'; ExternalWritable := 'False'} : Get_IM_Data;
   //    statGetImData2ErrorSaved { ExternalAccessible := 'False'; ExternalVisible := 'False'; ExternalWritable := 'False'} : Word := 16#0000;
   //    instGetImData3 { ExternalAccessible := 'False'; ExternalVisible := 'False'; ExternalWritable := 'False'} : Get_IM_Data;
   //    statGetImData3ErroSaved { ExternalAccessible := 'False'; ExternalVisible := 'False'; ExternalWritable := 'False'} : Word := 16#0000;
   //    instReadRecord { ExternalAccessible := 'False'; ExternalVisible := 'False'; ExternalWritable := 'False'} : RDREC;
   //    statReadRecordResult { ExternalAccessible := 'False'; ExternalVisible := 'False'; ExternalWritable := 'False'} : Array[0..199] of Byte;
   //    statStartNetAddresses { ExternalAccessible := 'False'; ExternalVisible := 'False'; ExternalWritable := 'False'} : USInt := 40;
   //    statIm1PlDesiLocIdLen { ExternalAccessible := 'False'; ExternalVisible := 'False'; ExternalWritable := 'False'} : Int := 54;
   //    statRisEdgeReadAll { ExternalAccessible := 'False'; ExternalVisible := 'False'; ExternalWritable := 'False'} : Bool := FALSE;
   //    statPosPulseReadAll { ExternalAccessible := 'False'; ExternalVisible := 'False'; ExternalWritable := 'False'} : Bool := FALSE;
   //    statErrorText { ExternalAccessible := 'False'; ExternalVisible := 'False'; ExternalWritable := 'False'} : String[30] := 'Error - Not readable data';
   // END_VAR
BEGIN
   instGetImData0.LADDR := 50;
   instGetImData0.IM_TYPE := 0;
   instGetImData0.DONE := TRUE;
   instGetImData0.BUSY := FALSE;
   instGetImData0.ERROR := FALSE;
   instGetImData0.STATUS := 16#0000;
   instGetImData0.sdw_GetAttrID := 16#0000_0031;
   instGetImData0.sdw_GetAttrAID := 16#0000_0EA9;
   instGetImData0.sdi_SfcLen := 60;
   instGetImData0.sb_useGetMultiAttr := FALSE;
   instGetImData0.sui_GetMultiAttrACount := 0;
   instGetImData0.sa_GetMultiAttrPathLens[0] := 0;
   instGetImData0.sa_GetMultiAttrPaths[0..2] := 0;
   instGetImData0.sa_GetMultiAttrResultLens[0] := 0;
   instGetImData0.sa_GetMultiAttrResult := ' ';
   instGetImData0.sb_SfcValid := TRUE;
   instGetImData0.sb_SfcERROR := FALSE;
   instGetImData0.sw_SfcStatus := 16#0000;
   instGetImData0.sa_SfcData[0] := 16#00;
   instGetImData0.sa_SfcData[1] := 16#20;
   instGetImData0.sa_SfcData[2] := 16#00;
   instGetImData0.sa_SfcData[3] := 16#38;
   instGetImData0.sa_SfcData[4] := 16#01;
   instGetImData0.sa_SfcData[5..6] := 16#00;
   instGetImData0.sa_SfcData[7] := 16#2A;
   instGetImData0.sa_SfcData[8] := 16#36;
   instGetImData0.sa_SfcData[9] := 16#45;
   instGetImData0.sa_SfcData[10] := 16#53;
   instGetImData0.sa_SfcData[11] := 16#37;
   instGetImData0.sa_SfcData[12] := 16#20;
   instGetImData0.sa_SfcData[13] := 16#35;
   instGetImData0.sa_SfcData[14] := 16#31;
   instGetImData0.sa_SfcData[15] := 16#38;
   instGetImData0.sa_SfcData[16] := 16#2D;
   instGetImData0.sa_SfcData[17] := 16#33;
   instGetImData0.sa_SfcData[18] := 16#55;
   instGetImData0.sa_SfcData[19] := 16#54;
   instGetImData0.sa_SfcData[20] := 16#31;
   instGetImData0.sa_SfcData[21] := 16#30;
   instGetImData0.sa_SfcData[22] := 16#2D;
   instGetImData0.sa_SfcData[23] := 16#30;
   instGetImData0.sa_SfcData[24] := 16#41;
   instGetImData0.sa_SfcData[25] := 16#42;
   instGetImData0.sa_SfcData[26] := 16#30;
   instGetImData0.sa_SfcData[27] := 16#20;
   instGetImData0.sa_SfcData[28] := 16#53;
   instGetImData0.sa_SfcData[29] := 16#20;
   instGetImData0.sa_SfcData[30] := 16#43;
   instGetImData0.sa_SfcData[31] := 16#2D;
   instGetImData0.sa_SfcData[32] := 16#54;
   instGetImData0.sa_SfcData[33] := 16#34;
   instGetImData0.sa_SfcData[34] := 16#41;
   instGetImData0.sa_SfcData[35] := 16#30;
   instGetImData0.sa_SfcData[36] := 16#52;
   instGetImData0.sa_SfcData[37] := 16#56;
   instGetImData0.sa_SfcData[38] := 16#48;
   instGetImData0.sa_SfcData[39] := 16#4D;
   instGetImData0.sa_SfcData[40] := 16#32;
   instGetImData0.sa_SfcData[41] := 16#30;
   instGetImData0.sa_SfcData[42] := 16#32;
   instGetImData0.sa_SfcData[43] := 16#35;
   instGetImData0.sa_SfcData[44] := 16#00;
   instGetImData0.sa_SfcData[45] := 16#01;
   instGetImData0.sa_SfcData[46] := 16#56;
   instGetImData0.sa_SfcData[47] := 16#04;
   instGetImData0.sa_SfcData[48..55] := 16#00;
   instGetImData0.sa_SfcData[56..57] := 16#01;
   instGetImData0.sa_SfcData[58] := 16#00;
   instGetImData0.sa_SfcData[59] := 16#0E;
   instGetImData0.sa_SfcData[60..64] := 16#00;
   instGetImData0.sudi_arraylength := 54;
   instGetImData0.sudi_datatype := 4;
   instGetImData0.sui_imdataLen := 54;
   instGetImData0.sui_imdataLen_netto := 54;
   instGetImData0.si_index := 16;
   instGetImData0.sb_SfcLocked := FALSE;
   instGetImData0.pw_TemporaryWord := 16#000E;
   instGetImData0.pa_DataByte[0..53] := 16#00;
   instGetImData0.pa_DataChar[0..53] := ' ';
   instGetImData0.pa_TemporaryCharArray[0] := 'S';
   instGetImData0.pa_TemporaryCharArray[1] := ' ';
   instGetImData0.pa_TemporaryCharArray[2] := 'C';
   instGetImData0.pa_TemporaryCharArray[3] := '-';
   instGetImData0.pa_TemporaryCharArray[4] := 'T';
   instGetImData0.pa_TemporaryCharArray[5] := '4';
   instGetImData0.pa_TemporaryCharArray[6] := 'A';
   instGetImData0.pa_TemporaryCharArray[7] := '0';
   instGetImData0.pa_TemporaryCharArray[8] := 'R';
   instGetImData0.pa_TemporaryCharArray[9] := 'V';
   instGetImData0.pa_TemporaryCharArray[10] := 'H';
   instGetImData0.pa_TemporaryCharArray[11] := 'M';
   instGetImData0.pa_TemporaryCharArray[12] := '2';
   instGetImData0.pa_TemporaryCharArray[13] := '0';
   instGetImData0.pa_TemporaryCharArray[14] := '2';
   instGetImData0.pa_TemporaryCharArray[15] := '5';
   instGetImData0.pa_TemporaryCharArray[16] := 'A';
   instGetImData0.pa_TemporaryCharArray[17] := 'B';
   instGetImData0.pa_TemporaryCharArray[18] := '0';
   instGetImData0.pa_TemporaryCharArray[19] := ' ';
   instGetImData0.p_DataUDT.Manufacturer_ID := 42;
   instGetImData0.p_DataUDT.Order_ID := '6ES7 518-3UT10-0AB0 ';
   instGetImData0.p_DataUDT.Serial_Number := 'S C-T4A0RVHM2025';
   instGetImData0.p_DataUDT.Hardware_Revision := 1;
   instGetImData0.p_DataUDT.Software_Revision."Type" := 'V';
   instGetImData0.p_DataUDT.Software_Revision.Functional := 4;
   instGetImData0.p_DataUDT.Software_Revision.Bugfix := 0;
   instGetImData0.p_DataUDT.Software_Revision.Internal := 0;
   instGetImData0.p_DataUDT.Revision_Counter := 0;
   instGetImData0.p_DataUDT.Profile_ID := 0;
   instGetImData0.p_DataUDT.Profile_Specific_Type := 0;
   instGetImData0.p_DataUDT.IM_Version := 16#0101;
   instGetImData0.p_DataUDT.IM_Supported := 16#000E;
   instGetImData1.LADDR := 50;
   instGetImData1.IM_TYPE := 11;
   instGetImData1.DONE := TRUE;
   instGetImData1.BUSY := FALSE;
   instGetImData1.ERROR := FALSE;
   instGetImData1.STATUS := 16#0000;
   instGetImData1.sdw_GetAttrID := 16#0000_0031;
   instGetImData1.sdw_GetAttrAID := 16#0000_0000;
   instGetImData1.sdi_SfcLen := 60;
   instGetImData1.sb_useGetMultiAttr := TRUE;
   instGetImData1.sui_GetMultiAttrACount := 1;
   instGetImData1.sa_GetMultiAttrPathLens[0] := 3;
   instGetImData1.sa_GetMultiAttrPaths[0] := 49;
   instGetImData1.sa_GetMultiAttrPaths[1] := 4690;
   instGetImData1.sa_GetMultiAttrPaths[2] := 45041;
   instGetImData1.sa_GetMultiAttrResultLens[0] := 0;
   instGetImData1.sa_GetMultiAttrResult := ' ';
   instGetImData1.sb_SfcValid := TRUE;
   instGetImData1.sb_SfcERROR := FALSE;
   instGetImData1.sw_SfcStatus := 16#0000;
   instGetImData1.sa_SfcData[0] := 16#00;
   instGetImData1.sa_SfcData[1] := 16#21;
   instGetImData1.sa_SfcData[2] := 16#00;
   instGetImData1.sa_SfcData[3] := 16#38;
   instGetImData1.sa_SfcData[4] := 16#01;
   instGetImData1.sa_SfcData[5] := 16#00;
   instGetImData1.sa_SfcData[6..59] := 16#20;
   instGetImData1.sa_SfcData[60..64] := 16#00;
   instGetImData1.sudi_arraylength := 0;
   instGetImData1.sudi_datatype := 1;
   instGetImData1.sui_imdataLen := 54;
   instGetImData1.sui_imdataLen_netto := 54;
   instGetImData1.si_index := 0;
   instGetImData1.sb_SfcLocked := FALSE;
   instGetImData1.pw_TemporaryWord := 16#0000;
   instGetImData1.pa_DataByte[0..53] := 16#00;
   instGetImData1.pa_DataChar[0..53] := ' ';
   instGetImData1.pa_TemporaryCharArray[0..19] := ' ';
   instGetImData1.p_DataUDT.Manufacturer_ID := 0;
   instGetImData1.p_DataUDT.Order_ID := '';
   instGetImData1.p_DataUDT.Serial_Number := '';
   instGetImData1.p_DataUDT.Hardware_Revision := 0;
   instGetImData1.p_DataUDT.Software_Revision."Type" := ' ';
   instGetImData1.p_DataUDT.Software_Revision.Functional := 0;
   instGetImData1.p_DataUDT.Software_Revision.Bugfix := 0;
   instGetImData1.p_DataUDT.Software_Revision.Internal := 0;
   instGetImData1.p_DataUDT.Revision_Counter := 0;
   instGetImData1.p_DataUDT.Profile_ID := 0;
   instGetImData1.p_DataUDT.Profile_Specific_Type := 0;
   instGetImData1.p_DataUDT.IM_Version := 16#0000;
   instGetImData1.p_DataUDT.IM_Supported := 16#0000;
   instGetImData2.LADDR := 50;
   instGetImData2.IM_TYPE := 12;
   instGetImData2.DONE := TRUE;
   instGetImData2.BUSY := FALSE;
   instGetImData2.ERROR := FALSE;
   instGetImData2.STATUS := 16#0000;
   instGetImData2.sdw_GetAttrID := 16#0000_0031;
   instGetImData2.sdw_GetAttrAID := 16#0000_0000;
   instGetImData2.sdi_SfcLen := 22;
   instGetImData2.sb_useGetMultiAttr := TRUE;
   instGetImData2.sui_GetMultiAttrACount := 1;
   instGetImData2.sa_GetMultiAttrPathLens[0] := 3;
   instGetImData2.sa_GetMultiAttrPaths[0] := 49;
   instGetImData2.sa_GetMultiAttrPaths[1] := 4690;
   instGetImData2.sa_GetMultiAttrPaths[2] := 45042;
   instGetImData2.sa_GetMultiAttrResultLens[0] := 0;
   instGetImData2.sa_GetMultiAttrResult := ' ';
   instGetImData2.sb_SfcValid := TRUE;
   instGetImData2.sb_SfcERROR := FALSE;
   instGetImData2.sw_SfcStatus := 16#0000;
   instGetImData2.sa_SfcData[0] := 16#00;
   instGetImData2.sa_SfcData[1] := 16#22;
   instGetImData2.sa_SfcData[2] := 16#00;
   instGetImData2.sa_SfcData[3] := 16#12;
   instGetImData2.sa_SfcData[4] := 16#01;
   instGetImData2.sa_SfcData[5] := 16#00;
   instGetImData2.sa_SfcData[6] := 16#32;
   instGetImData2.sa_SfcData[7] := 16#30;
   instGetImData2.sa_SfcData[8] := 16#32;
   instGetImData2.sa_SfcData[9] := 16#35;
   instGetImData2.sa_SfcData[10] := 16#2D;
   instGetImData2.sa_SfcData[11] := 16#30;
   instGetImData2.sa_SfcData[12] := 16#32;
   instGetImData2.sa_SfcData[13] := 16#2D;
   instGetImData2.sa_SfcData[14] := 16#32;
   instGetImData2.sa_SfcData[15] := 16#34;
   instGetImData2.sa_SfcData[16] := 16#20;
   instGetImData2.sa_SfcData[17] := 16#31;
   instGetImData2.sa_SfcData[18] := 16#36;
   instGetImData2.sa_SfcData[19] := 16#3A;
   instGetImData2.sa_SfcData[20] := 16#35;
   instGetImData2.sa_SfcData[21] := 16#39;
   instGetImData2.sa_SfcData[22..64] := 16#00;
   instGetImData2.sudi_arraylength := 0;
   instGetImData2.sudi_datatype := 1;
   instGetImData2.sui_imdataLen := 16;
   instGetImData2.sui_imdataLen_netto := 16;
   instGetImData2.si_index := 0;
   instGetImData2.sb_SfcLocked := FALSE;
   instGetImData2.pw_TemporaryWord := 16#0000;
   instGetImData2.pa_DataByte[0..53] := 16#00;
   instGetImData2.pa_DataChar[0..53] := ' ';
   instGetImData2.pa_TemporaryCharArray[0..19] := ' ';
   instGetImData2.p_DataUDT.Manufacturer_ID := 0;
   instGetImData2.p_DataUDT.Order_ID := '';
   instGetImData2.p_DataUDT.Serial_Number := '';
   instGetImData2.p_DataUDT.Hardware_Revision := 0;
   instGetImData2.p_DataUDT.Software_Revision."Type" := ' ';
   instGetImData2.p_DataUDT.Software_Revision.Functional := 0;
   instGetImData2.p_DataUDT.Software_Revision.Bugfix := 0;
   instGetImData2.p_DataUDT.Software_Revision.Internal := 0;
   instGetImData2.p_DataUDT.Revision_Counter := 0;
   instGetImData2.p_DataUDT.Profile_ID := 0;
   instGetImData2.p_DataUDT.Profile_Specific_Type := 0;
   instGetImData2.p_DataUDT.IM_Version := 16#0000;
   instGetImData2.p_DataUDT.IM_Supported := 16#0000;
   instGetImData3.LADDR := 50;
   instGetImData3.IM_TYPE := 13;
   instGetImData3.DONE := TRUE;
   instGetImData3.BUSY := FALSE;
   instGetImData3.ERROR := FALSE;
   instGetImData3.STATUS := 16#0000;
   instGetImData3.sdw_GetAttrID := 16#0000_0031;
   instGetImData3.sdw_GetAttrAID := 16#0000_0000;
   instGetImData3.sdi_SfcLen := 60;
   instGetImData3.sb_useGetMultiAttr := TRUE;
   instGetImData3.sui_GetMultiAttrACount := 1;
   instGetImData3.sa_GetMultiAttrPathLens[0] := 3;
   instGetImData3.sa_GetMultiAttrPaths[0] := 49;
   instGetImData3.sa_GetMultiAttrPaths[1] := 4690;
   instGetImData3.sa_GetMultiAttrPaths[2] := 45043;
   instGetImData3.sa_GetMultiAttrResultLens[0] := 0;
   instGetImData3.sa_GetMultiAttrResult := ' ';
   instGetImData3.sb_SfcValid := TRUE;
   instGetImData3.sb_SfcERROR := FALSE;
   instGetImData3.sw_SfcStatus := 16#0000;
   instGetImData3.sa_SfcData[0] := 16#00;
   instGetImData3.sa_SfcData[1] := 16#23;
   instGetImData3.sa_SfcData[2] := 16#00;
   instGetImData3.sa_SfcData[3] := 16#38;
   instGetImData3.sa_SfcData[4] := 16#01;
   instGetImData3.sa_SfcData[5] := 16#00;
   instGetImData3.sa_SfcData[6..59] := 16#20;
   instGetImData3.sa_SfcData[60..64] := 16#00;
   instGetImData3.sudi_arraylength := 0;
   instGetImData3.sudi_datatype := 1;
   instGetImData3.sui_imdataLen := 54;
   instGetImData3.sui_imdataLen_netto := 54;
   instGetImData3.si_index := 0;
   instGetImData3.sb_SfcLocked := FALSE;
   instGetImData3.pw_TemporaryWord := 16#0000;
   instGetImData3.pa_DataByte[0..53] := 16#00;
   instGetImData3.pa_DataChar[0..53] := ' ';
   instGetImData3.pa_TemporaryCharArray[0..19] := ' ';
   instGetImData3.p_DataUDT.Manufacturer_ID := 0;
   instGetImData3.p_DataUDT.Order_ID := '';
   instGetImData3.p_DataUDT.Serial_Number := '';
   instGetImData3.p_DataUDT.Hardware_Revision := 0;
   instGetImData3.p_DataUDT.Software_Revision."Type" := ' ';
   instGetImData3.p_DataUDT.Software_Revision.Functional := 0;
   instGetImData3.p_DataUDT.Software_Revision.Bugfix := 0;
   instGetImData3.p_DataUDT.Software_Revision.Internal := 0;
   instGetImData3.p_DataUDT.Revision_Counter := 0;
   instGetImData3.p_DataUDT.Profile_ID := 0;
   instGetImData3.p_DataUDT.Profile_Specific_Type := 0;
   instGetImData3.p_DataUDT.IM_Version := 16#0000;
   instGetImData3.p_DataUDT.IM_Supported := 16#0000;
   instReadRecord.REQ := FALSE;
   instReadRecord.ID := 64;
   instReadRecord.INDEX := 32896;
   instReadRecord.MLEN := 200;
   instReadRecord.VALID := FALSE;
   instReadRecord.BUSY := FALSE;
   instReadRecord.ERROR := FALSE;
   instReadRecord.STATUS := 16#0070_0000;
   instReadRecord.LEN := 0;
   statReadRecordResult[0] := 16#02;
   statReadRecordResult[1] := 16#40;
   statReadRecordResult[2] := 16#00;
   statReadRecordResult[3] := 16#38;
   statReadRecordResult[4] := 16#01;
   statReadRecordResult[5] := 16#00;
   statReadRecordResult[6] := 16#1E;
   statReadRecordResult[7] := 16#62;
   statReadRecordResult[8] := 16#61;
   statReadRecordResult[9] := 16#30;
   statReadRecordResult[10] := 16#33;
   statReadRecordResult[11] := 16#30;
   statReadRecordResult[12] := 16#61;
   statReadRecordResult[13] := 16#7A;
   statReadRecordResult[14] := 16#73;
   statReadRecordResult[15] := 16#63;
   statReadRecordResult[16] := 16#31;
   statReadRecordResult[17] := 16#2E;
   statReadRecordResult[18] := 16#62;
   statReadRecordResult[19] := 16#61;
   statReadRecordResult[20] := 16#30;
   statReadRecordResult[21] := 16#33;
   statReadRecordResult[22] := 16#30;
   statReadRecordResult[23] := 16#61;
   statReadRecordResult[24] := 16#7A;
   statReadRecordResult[25] := 16#73;
   statReadRecordResult[26] := 16#63;
   statReadRecordResult[27] := 16#31;
   statReadRecordResult[28] := 16#78;
   statReadRecordResult[29] := 16#62;
   statReadRecordResult[30..31] := 16#78;
   statReadRecordResult[32] := 16#31;
   statReadRecordResult[33] := 16#33;
   statReadRecordResult[34] := 16#63;
   statReadRecordResult[35] := 16#33;
   statReadRecordResult[36] := 16#66;
   statReadRecordResult[37..39] := 16#00;
   statReadRecordResult[40] := 16#30;
   statReadRecordResult[41] := 16#B8;
   statReadRecordResult[42] := 16#51;
   statReadRecordResult[43] := 16#66;
   statReadRecordResult[44] := 16#CF;
   statReadRecordResult[45] := 16#66;
   statReadRecordResult[46..47] := 16#00;
   statReadRecordResult[48] := 16#C0;
   statReadRecordResult[49] := 16#A8;
   statReadRecordResult[50] := 16#C8;
   statReadRecordResult[51] := 16#33;
   statReadRecordResult[52..54] := 16#FF;
   statReadRecordResult[55] := 16#00;
   statReadRecordResult[56] := 16#C0;
   statReadRecordResult[57] := 16#A8;
   statReadRecordResult[58] := 16#C8;
   statReadRecordResult[59] := 16#33;
   statReadRecordResult[60..199] := 16#00;
END_DATA_BLOCK

DATA_BLOCK "IdentRfInterfaceHmi"   // DB218
// stored: InstanceOfName typeIdentRfHmi, InstanceOfType UDT
"typeIdentRfHmi"
BEGIN
   rfReader[0..1].deviceName := WSTRING#'';
   rfReader[0..1].deviceType := WSTRING#'';
   rfReader[0..1].deviceId := 0;
   rfReader[0..1].tagType := WSTRING#'';
   rfReader[0..1].cameraMode := WSTRING#'';
   rfReader[0..1].resultState := WSTRING#'';
   rfReader[0..1].progNo := 0;
   rfReader[0..1].progNumberWrite := 0;
   rfReader[0..1].pushbutton := 16#0000;
   rfReader[0..1].enablePushbutton := 16#0000;
   rfReader[0..1].status := 16#0000;
   rfReader[0..1].alarmCategorie := 0;
   rfReader[0..1].alarmNo := 0;
   rfReader[0..1].alarmCode := 16#0000_0000;
   rfReader[0..1].resultColor := 0;
   rfReader[0..1].statusColorCode := 0;
   rfReader[0..1].datRead1 := '';
   rfReader[0..1].datRead2 := '';
   rfReader[0..1].datRead3 := '';
   rfReader[0..1].datRead4 := '';
   rfReader[0..1].datWrite1 := '';
   rfReader[0..1].datWrite2 := '';
   rfReader[0..1].datWrite3 := '';
   rfReader[0..1].datWrite4 := '';
END_DATA_BLOCK

DATA_BLOCK "instGetIdentRf"   // DB217
// stored: InstanceOfName GetIdentRf, InstanceOfType FB
"GetIdentRf"
BEGIN
   identRfAllUnits[0].identRfEM[0..7].selectedUnit := 0;
   identRfAllUnits[0].identRfEM[0..7].selectedEM := 0;
   identRfAllUnits[0].identRfEM[0..7].rfReaderId := 0;
   identRfAllUnits[0].identRfEM[0..7].numberOfRf := 0;
   identRfAllUnits[0].identRfEM[0].rfReader[0..1].deviceName := WSTRING#'';
   identRfAllUnits[0].identRfEM[1].rfReader[0..1].deviceName := WSTRING#'';
   identRfAllUnits[0].identRfEM[2].rfReader[0..1].deviceName := WSTRING#'';
   identRfAllUnits[0].identRfEM[3].rfReader[0..1].deviceName := WSTRING#'';
   identRfAllUnits[0].identRfEM[4].rfReader[0..1].deviceName := WSTRING#'';
   identRfAllUnits[0].identRfEM[5].rfReader[0..1].deviceName := WSTRING#'';
   identRfAllUnits[0].identRfEM[6].rfReader[0..1].deviceName := WSTRING#'';
   identRfAllUnits[0].identRfEM[7].rfReader[0..1].deviceName := WSTRING#'';
   identRfAllUnits[0].identRfEM[0].rfReader[0..1].deviceType := WSTRING#'';
   identRfAllUnits[0].identRfEM[1].rfReader[0..1].deviceType := WSTRING#'';
   identRfAllUnits[0].identRfEM[2].rfReader[0..1].deviceType := WSTRING#'';
   identRfAllUnits[0].identRfEM[3].rfReader[0..1].deviceType := WSTRING#'';
   identRfAllUnits[0].identRfEM[4].rfReader[0..1].deviceType := WSTRING#'';
   identRfAllUnits[0].identRfEM[5].rfReader[0..1].deviceType := WSTRING#'';
   identRfAllUnits[0].identRfEM[6].rfReader[0..1].deviceType := WSTRING#'';
   identRfAllUnits[0].identRfEM[7].rfReader[0..1].deviceType := WSTRING#'';
   identRfAllUnits[0].identRfEM[0].rfReader[0..1].deviceId := 0;
   identRfAllUnits[0].identRfEM[1].rfReader[0..1].deviceId := 0;
   identRfAllUnits[0].identRfEM[2].rfReader[0..1].deviceId := 0;
   identRfAllUnits[0].identRfEM[3].rfReader[0..1].deviceId := 0;
   identRfAllUnits[0].identRfEM[4].rfReader[0..1].deviceId := 0;
   identRfAllUnits[0].identRfEM[5].rfReader[0..1].deviceId := 0;
   identRfAllUnits[0].identRfEM[6].rfReader[0..1].deviceId := 0;
   identRfAllUnits[0].identRfEM[7].rfReader[0..1].deviceId := 0;
   identRfAllUnits[0].identRfEM[0].rfReader[0..1].tagType := WSTRING#'';
   identRfAllUnits[0].identRfEM[1].rfReader[0..1].tagType := WSTRING#'';
   identRfAllUnits[0].identRfEM[2].rfReader[0..1].tagType := WSTRING#'';
   identRfAllUnits[0].identRfEM[3].rfReader[0..1].tagType := WSTRING#'';
   identRfAllUnits[0].identRfEM[4].rfReader[0..1].tagType := WSTRING#'';
   identRfAllUnits[0].identRfEM[5].rfReader[0..1].tagType := WSTRING#'';
   identRfAllUnits[0].identRfEM[6].rfReader[0..1].tagType := WSTRING#'';
   identRfAllUnits[0].identRfEM[7].rfReader[0..1].tagType := WSTRING#'';
   identRfAllUnits[0].identRfEM[0].rfReader[0..1].cameraMode := WSTRING#'';
   identRfAllUnits[0].identRfEM[1].rfReader[0..1].cameraMode := WSTRING#'';
   identRfAllUnits[0].identRfEM[2].rfReader[0..1].cameraMode := WSTRING#'';
   identRfAllUnits[0].identRfEM[3].rfReader[0..1].cameraMode := WSTRING#'';
   identRfAllUnits[0].identRfEM[4].rfReader[0..1].cameraMode := WSTRING#'';
   identRfAllUnits[0].identRfEM[5].rfReader[0..1].cameraMode := WSTRING#'';
   identRfAllUnits[0].identRfEM[6].rfReader[0..1].cameraMode := WSTRING#'';
   identRfAllUnits[0].identRfEM[7].rfReader[0..1].cameraMode := WSTRING#'';
   identRfAllUnits[0].identRfEM[0].rfReader[0..1].resultState := WSTRING#'';
   identRfAllUnits[0].identRfEM[1].rfReader[0..1].resultState := WSTRING#'';
   identRfAllUnits[0].identRfEM[2].rfReader[0..1].resultState := WSTRING#'';
   identRfAllUnits[0].identRfEM[3].rfReader[0..1].resultState := WSTRING#'';
   identRfAllUnits[0].identRfEM[4].rfReader[0..1].resultState := WSTRING#'';
   identRfAllUnits[0].identRfEM[5].rfReader[0..1].resultState := WSTRING#'';
   identRfAllUnits[0].identRfEM[6].rfReader[0..1].resultState := WSTRING#'';
   identRfAllUnits[0].identRfEM[7].rfReader[0..1].resultState := WSTRING#'';
   identRfAllUnits[0].identRfEM[0].rfReader[0..1].progNo := 0;
   identRfAllUnits[0].identRfEM[1].rfReader[0..1].progNo := 0;
   identRfAllUnits[0].identRfEM[2].rfReader[0..1].progNo := 0;
   identRfAllUnits[0].identRfEM[3].rfReader[0..1].progNo := 0;
   identRfAllUnits[0].identRfEM[4].rfReader[0..1].progNo := 0;
   identRfAllUnits[0].identRfEM[5].rfReader[0..1].progNo := 0;
   identRfAllUnits[0].identRfEM[6].rfReader[0..1].progNo := 0;
   identRfAllUnits[0].identRfEM[7].rfReader[0..1].progNo := 0;
   identRfAllUnits[0].identRfEM[0].rfReader[0..1].progNumberWrite := 0;
   identRfAllUnits[0].identRfEM[1].rfReader[0..1].progNumberWrite := 0;
   identRfAllUnits[0].identRfEM[2].rfReader[0..1].progNumberWrite := 0;
   identRfAllUnits[0].identRfEM[3].rfReader[0..1].progNumberWrite := 0;
   identRfAllUnits[0].identRfEM[4].rfReader[0..1].progNumberWrite := 0;
   identRfAllUnits[0].identRfEM[5].rfReader[0..1].progNumberWrite := 0;
   identRfAllUnits[0].identRfEM[6].rfReader[0..1].progNumberWrite := 0;
   identRfAllUnits[0].identRfEM[7].rfReader[0..1].progNumberWrite := 0;
   identRfAllUnits[0].identRfEM[0].rfReader[0..1].pushbutton := 16#0000;
   identRfAllUnits[0].identRfEM[1].rfReader[0..1].pushbutton := 16#0000;
   identRfAllUnits[0].identRfEM[2].rfReader[0..1].pushbutton := 16#0000;
   identRfAllUnits[0].identRfEM[3].rfReader[0..1].pushbutton := 16#0000;
   identRfAllUnits[0].identRfEM[4].rfReader[0..1].pushbutton := 16#0000;
   identRfAllUnits[0].identRfEM[5].rfReader[0..1].pushbutton := 16#0000;
   identRfAllUnits[0].identRfEM[6].rfReader[0..1].pushbutton := 16#0000;
   identRfAllUnits[0].identRfEM[7].rfReader[0..1].pushbutton := 16#0000;
   identRfAllUnits[0].identRfEM[0].rfReader[0..1].enablePushbutton := 16#0000;
   identRfAllUnits[0].identRfEM[1].rfReader[0..1].enablePushbutton := 16#0000;
   identRfAllUnits[0].identRfEM[2].rfReader[0..1].enablePushbutton := 16#0000;
   identRfAllUnits[0].identRfEM[3].rfReader[0..1].enablePushbutton := 16#0000;
   identRfAllUnits[0].identRfEM[4].rfReader[0..1].enablePushbutton := 16#0000;
   identRfAllUnits[0].identRfEM[5].rfReader[0..1].enablePushbutton := 16#0000;
   identRfAllUnits[0].identRfEM[6].rfReader[0..1].enablePushbutton := 16#0000;
   identRfAllUnits[0].identRfEM[7].rfReader[0..1].enablePushbutton := 16#0000;
   identRfAllUnits[0].identRfEM[0].rfReader[0..1].status := 16#0000;
   identRfAllUnits[0].identRfEM[1].rfReader[0..1].status := 16#0000;
   identRfAllUnits[0].identRfEM[2].rfReader[0..1].status := 16#0000;
   identRfAllUnits[0].identRfEM[3].rfReader[0..1].status := 16#0000;
   identRfAllUnits[0].identRfEM[4].rfReader[0..1].status := 16#0000;
   identRfAllUnits[0].identRfEM[5].rfReader[0..1].status := 16#0000;
   identRfAllUnits[0].identRfEM[6].rfReader[0..1].status := 16#0000;
   identRfAllUnits[0].identRfEM[7].rfReader[0..1].status := 16#0000;
   identRfAllUnits[0].identRfEM[0].rfReader[0..1].alarmCategorie := 0;
   identRfAllUnits[0].identRfEM[1].rfReader[0..1].alarmCategorie := 0;
   identRfAllUnits[0].identRfEM[2].rfReader[0..1].alarmCategorie := 0;
   identRfAllUnits[0].identRfEM[3].rfReader[0..1].alarmCategorie := 0;
   identRfAllUnits[0].identRfEM[4].rfReader[0..1].alarmCategorie := 0;
   identRfAllUnits[0].identRfEM[5].rfReader[0..1].alarmCategorie := 0;
   identRfAllUnits[0].identRfEM[6].rfReader[0..1].alarmCategorie := 0;
   identRfAllUnits[0].identRfEM[7].rfReader[0..1].alarmCategorie := 0;
   identRfAllUnits[0].identRfEM[0].rfReader[0..1].alarmNo := 0;
   identRfAllUnits[0].identRfEM[1].rfReader[0..1].alarmNo := 0;
   identRfAllUnits[0].identRfEM[2].rfReader[0..1].alarmNo := 0;
   identRfAllUnits[0].identRfEM[3].rfReader[0..1].alarmNo := 0;
   identRfAllUnits[0].identRfEM[4].rfReader[0..1].alarmNo := 0;
   identRfAllUnits[0].identRfEM[5].rfReader[0..1].alarmNo := 0;
   identRfAllUnits[0].identRfEM[6].rfReader[0..1].alarmNo := 0;
   identRfAllUnits[0].identRfEM[7].rfReader[0..1].alarmNo := 0;
   identRfAllUnits[0].identRfEM[0].rfReader[0..1].alarmCode := 16#0000_0000;
   identRfAllUnits[0].identRfEM[1].rfReader[0..1].alarmCode := 16#0000_0000;
   identRfAllUnits[0].identRfEM[2].rfReader[0..1].alarmCode := 16#0000_0000;
   identRfAllUnits[0].identRfEM[3].rfReader[0..1].alarmCode := 16#0000_0000;
   identRfAllUnits[0].identRfEM[4].rfReader[0..1].alarmCode := 16#0000_0000;
   identRfAllUnits[0].identRfEM[5].rfReader[0..1].alarmCode := 16#0000_0000;
   identRfAllUnits[0].identRfEM[6].rfReader[0..1].alarmCode := 16#0000_0000;
   identRfAllUnits[0].identRfEM[7].rfReader[0..1].alarmCode := 16#0000_0000;
   identRfAllUnits[0].identRfEM[0].rfReader[0..1].resultColor := 0;
   identRfAllUnits[0].identRfEM[1].rfReader[0..1].resultColor := 0;
   identRfAllUnits[0].identRfEM[2].rfReader[0..1].resultColor := 0;
   identRfAllUnits[0].identRfEM[3].rfReader[0..1].resultColor := 0;
   identRfAllUnits[0].identRfEM[4].rfReader[0..1].resultColor := 0;
   identRfAllUnits[0].identRfEM[5].rfReader[0..1].resultColor := 0;
   identRfAllUnits[0].identRfEM[6].rfReader[0..1].resultColor := 0;
   identRfAllUnits[0].identRfEM[7].rfReader[0..1].resultColor := 0;
   identRfAllUnits[0].identRfEM[0].rfReader[0..1].statusColorCode := 0;
   identRfAllUnits[0].identRfEM[1].rfReader[0..1].statusColorCode := 0;
   identRfAllUnits[0].identRfEM[2].rfReader[0..1].statusColorCode := 0;
   identRfAllUnits[0].identRfEM[3].rfReader[0..1].statusColorCode := 0;
   identRfAllUnits[0].identRfEM[4].rfReader[0..1].statusColorCode := 0;
   identRfAllUnits[0].identRfEM[5].rfReader[0..1].statusColorCode := 0;
   identRfAllUnits[0].identRfEM[6].rfReader[0..1].statusColorCode := 0;
   identRfAllUnits[0].identRfEM[7].rfReader[0..1].statusColorCode := 0;
   identRfAllUnits[0].identRfEM[0].rfReader[0..1].datRead1 := '';
   identRfAllUnits[0].identRfEM[1].rfReader[0..1].datRead1 := '';
   identRfAllUnits[0].identRfEM[2].rfReader[0..1].datRead1 := '';
   identRfAllUnits[0].identRfEM[3].rfReader[0..1].datRead1 := '';
   identRfAllUnits[0].identRfEM[4].rfReader[0..1].datRead1 := '';
   identRfAllUnits[0].identRfEM[5].rfReader[0..1].datRead1 := '';
   identRfAllUnits[0].identRfEM[6].rfReader[0..1].datRead1 := '';
   identRfAllUnits[0].identRfEM[7].rfReader[0..1].datRead1 := '';
   identRfAllUnits[0].identRfEM[0].rfReader[0..1].datRead2 := '';
   identRfAllUnits[0].identRfEM[1].rfReader[0..1].datRead2 := '';
   identRfAllUnits[0].identRfEM[2].rfReader[0..1].datRead2 := '';
   identRfAllUnits[0].identRfEM[3].rfReader[0..1].datRead2 := '';
   identRfAllUnits[0].identRfEM[4].rfReader[0..1].datRead2 := '';
   identRfAllUnits[0].identRfEM[5].rfReader[0..1].datRead2 := '';
   identRfAllUnits[0].identRfEM[6].rfReader[0..1].datRead2 := '';
   identRfAllUnits[0].identRfEM[7].rfReader[0..1].datRead2 := '';
   identRfAllUnits[0].identRfEM[0].rfReader[0..1].datRead3 := '';
   identRfAllUnits[0].identRfEM[1].rfReader[0..1].datRead3 := '';
   identRfAllUnits[0].identRfEM[2].rfReader[0..1].datRead3 := '';
   identRfAllUnits[0].identRfEM[3].rfReader[0..1].datRead3 := '';
   identRfAllUnits[0].identRfEM[4].rfReader[0..1].datRead3 := '';
   identRfAllUnits[0].identRfEM[5].rfReader[0..1].datRead3 := '';
   identRfAllUnits[0].identRfEM[6].rfReader[0..1].datRead3 := '';
   identRfAllUnits[0].identRfEM[7].rfReader[0..1].datRead3 := '';
   identRfAllUnits[0].identRfEM[0].rfReader[0..1].datRead4 := '';
   identRfAllUnits[0].identRfEM[1].rfReader[0..1].datRead4 := '';
   identRfAllUnits[0].identRfEM[2].rfReader[0..1].datRead4 := '';
   identRfAllUnits[0].identRfEM[3].rfReader[0..1].datRead4 := '';
   identRfAllUnits[0].identRfEM[4].rfReader[0..1].datRead4 := '';
   identRfAllUnits[0].identRfEM[5].rfReader[0..1].datRead4 := '';
   identRfAllUnits[0].identRfEM[6].rfReader[0..1].datRead4 := '';
   identRfAllUnits[0].identRfEM[7].rfReader[0..1].datRead4 := '';
   identRfAllUnits[0].identRfEM[0].rfReader[0..1].datWrite1 := '';
   identRfAllUnits[0].identRfEM[1].rfReader[0..1].datWrite1 := '';
   identRfAllUnits[0].identRfEM[2].rfReader[0..1].datWrite1 := '';
   identRfAllUnits[0].identRfEM[3].rfReader[0..1].datWrite1 := '';
   identRfAllUnits[0].identRfEM[4].rfReader[0..1].datWrite1 := '';
   identRfAllUnits[0].identRfEM[5].rfReader[0..1].datWrite1 := '';
   identRfAllUnits[0].identRfEM[6].rfReader[0..1].datWrite1 := '';
   identRfAllUnits[0].identRfEM[7].rfReader[0..1].datWrite1 := '';
   identRfAllUnits[0].identRfEM[0].rfReader[0..1].datWrite2 := '';
   identRfAllUnits[0].identRfEM[1].rfReader[0..1].datWrite2 := '';
   identRfAllUnits[0].identRfEM[2].rfReader[0..1].datWrite2 := '';
   identRfAllUnits[0].identRfEM[3].rfReader[0..1].datWrite2 := '';
   identRfAllUnits[0].identRfEM[4].rfReader[0..1].datWrite2 := '';
   identRfAllUnits[0].identRfEM[5].rfReader[0..1].datWrite2 := '';
   identRfAllUnits[0].identRfEM[6].rfReader[0..1].datWrite2 := '';
   identRfAllUnits[0].identRfEM[7].rfReader[0..1].datWrite2 := '';
   identRfAllUnits[0].identRfEM[0].rfReader[0..1].datWrite3 := '';
   identRfAllUnits[0].identRfEM[1].rfReader[0..1].datWrite3 := '';
   identRfAllUnits[0].identRfEM[2].rfReader[0..1].datWrite3 := '';
   identRfAllUnits[0].identRfEM[3].rfReader[0..1].datWrite3 := '';
   identRfAllUnits[0].identRfEM[4].rfReader[0..1].datWrite3 := '';
   identRfAllUnits[0].identRfEM[5].rfReader[0..1].datWrite3 := '';
   identRfAllUnits[0].identRfEM[6].rfReader[0..1].datWrite3 := '';
   identRfAllUnits[0].identRfEM[7].rfReader[0..1].datWrite3 := '';
   identRfAllUnits[0].identRfEM[0].rfReader[0..1].datWrite4 := '';
   identRfAllUnits[0].identRfEM[1].rfReader[0..1].datWrite4 := '';
   identRfAllUnits[0].identRfEM[2].rfReader[0..1].datWrite4 := '';
   identRfAllUnits[0].identRfEM[3].rfReader[0..1].datWrite4 := '';
   identRfAllUnits[0].identRfEM[4].rfReader[0..1].datWrite4 := '';
   identRfAllUnits[0].identRfEM[5].rfReader[0..1].datWrite4 := '';
   identRfAllUnits[0].identRfEM[6].rfReader[0..1].datWrite4 := '';
   identRfAllUnits[0].identRfEM[7].rfReader[0..1].datWrite4 := '';
END_DATA_BLOCK

DATA_BLOCK "IdentMvInterfaceHmi"   // DB219
// stored: InstanceOfName typeIdentMvHmi, InstanceOfType UDT
"typeIdentMvHmi"
BEGIN
   mvReader[0..1].deviceName := WSTRING#'';
   mvReader[0..1].deviceType := WSTRING#'';
   mvReader[0..1].deviceId := 0;
   mvReader[0..1].tagType := WSTRING#'';
   mvReader[0..1].cameraMode := WSTRING#'';
   mvReader[0..1].resultState := WSTRING#'';
   mvReader[0..1].progNo := 0;
   mvReader[0..1].progNumberWrite := 0;
   mvReader[0..1].pushbutton := 16#0000;
   mvReader[0..1].enablePushbutton := 16#0000;
   mvReader[0..1].status := 16#0000;
   mvReader[0..1].alarmCategorie := 0;
   mvReader[0..1].alarmNo := 0;
   mvReader[0..1].alarmCode := 16#0000_0000;
   mvReader[0..1].resultColor := 0;
   mvReader[0..1].statusColorCode := 0;
   mvReader[0..1].datRead1 := '';
   mvReader[0..1].datRead2 := '';
   mvReader[0..1].datRead3 := '';
   mvReader[0..1].datRead4 := '';
   mvReader[0..1].datWrite1 := '';
   mvReader[0..1].datWrite2 := '';
   mvReader[0..1].datWrite3 := '';
   mvReader[0..1].datWrite4 := '';
END_DATA_BLOCK

